(* CODESYS project gprs.lock.20190507.1.project

Project tree, tasks and I/O mapping:
  MIC7001 : Changsha Xiangji-ARM Cortex A9(xilinx zynq7000)-linux, Changsha Xiangji Hiden Technology Co.Ltd, version 3.5.10.40
    application Application
      libraries: Standard, * (System); CAA File, * (CAA Technical Workgroup); CAA Types Extern, * (CAA Technical Workgroup); CAA Callback Extern, * (CAA Technical Workgroup); SysMem, * (System); Util, 3.5.11.0 (System); SysFile, 3.5.9.0 (System); SysTypes Interfaces, * (System); CAN API, 1.0.0.3 (3S - Smart Software Solutions GmbH); AC_DataLog, 3.5.12.0 (3S - Smart Software Solutions GmbH); SysTime, * (System); CAA DTUtil Extern, 3.5.12.0 (CAA Technical Workgroup); CAA SerialCom, 3.5.12.0 (CAA Technical Workgroup); cyber gpio, 3.5.10.40 (cyber)
      task Task_gprs (cyclic, interval 20 ms, priority 10) calls prg_heartbeat
      gprs_lib/
        function block Udp_Config [ST]
        function block reset_gprs [ST]
        function block Udp_Init [ST]
        function block Com_Read [ST]
        function block UDP_Read [ST]
        function block Udp_Write [ST]
      global variables GVL
      GPRS/
        function block fb_get_lac [ST]
        function block fb_get_iccid [ST]
        program prg_heartbeat [ST]
        function block File_Read [ST]
        function block fb_m26 [ST]
        function fn_sn_str_to_byte [ST]
        function Iccid_Get [ST]
        function fn_cyber_layer1 [ST]
        function fn_cyber_userdata200 [ST]
        function fn_cyber_layer2 [ST]
        function fn_cyber_heartBeat [ST]
    SoftMotion General Axis Pool
    IoDrvMIC7001 : IoDrvMIC7001, MyCompany, version 19.1.1
        input  Application.GVL.FR_Protect_DI : BOOL  // Di00-Ai00@C16
        input  Application.GVL.PumpOn_DI : BOOL  // Di01-Ai01@C28
        input  Application.GVL.Remot_Enable_DI : BOOL  // Di02-Ai02@C17
        input  Application.GVL.Rev_PumpOn_DI : BOOL  // Di03-Ai03@C29
        input  Application.GVL.LeftZG_Forward_DI : BOOL  // Di04-Ai04@C30
        input  Application.GVL.Flux_Down_DI : BOOL  // Di05-Ai05@C19
        input  Application.GVL.RightZG_Forward_DI : BOOL  // Di06-Ai06@C31
        input  Application.GVL.ADDOn_DI : BOOL  // Di07-Ai07@C20
        input  Application.GVL.Flux_Up_DI : BOOL  // Di08-Ai08@C18
        input  Application.GVL.Leg_BG_DI : BOOL  // Di09-Ai09@D18
        input  Application.GVL.Limit_Right_DI : BOOL  // Di10-Ai10@D20
        input  Application.GVL.AC_Power_DI : BOOL  // Di11-Ai11@D31
        input  Application.GVL.Limit_Left_DI : BOOL  // Di12-Ai12@D19
        input  Application.GVL.Power_Order_DI : BOOL  // Di14-Ai14@D29
        input  Application.GVL.LeftBG_Forward_DI : BOOL  // Di15-Ai15@D17
        input  Application.GVL.Right_SQ_DI : BOOL  // Di16-Ai16@D28
        input  Application.GVL.RightBG_Forward_DI : BOOL  // Di17-Ai17@D16
        input  Application.GVL.DI_move : BOOL  // Di27-Ai27@C09
        input  Application.GVL.ADDFlux_Down_DI : BOOL  // Di46-Ai46@C22
        input  Application.GVL.ADDFlux_Up_DI : BOOL  // Di47-Ai47@D14
        input  Application.GVL.Motor_Stop_DI : BOOL  // Di48-Pi00@C15
        input  Application.GVL.Motor_Start_DI : BOOL  // Di49-Pi01@C14
        input  Application.GVL.Left_SQ_DI : BOOL  // Di50-Pi02@D22
        input  Application.GVL.Light_Boom_DI : BOOL  // Di51-Pi03@D21
        output Application.GVL.ERR_Power_Order : BOOL  // Do00-Ai18@C25
        output Application.GVL.Remot_Control_DO : BOOL  // Do01-Ai19@C24
        output Application.GVL.Alarm_DO : BOOL  // Do02-Ai20@C13
        output Application.GVL.Light_Boom_DO : BOOL  // Do03-Ai21@C01
        output Application.GVL.DT2_DO : BOOL  // Do04-Ai22@C03
        output Application.GVL.DT3_DO : BOOL  // Do05-Ai23@C04
        output Application.GVL.DT5_DO : BOOL  // Do06-Ai24@C05
        output Application.GVL.DT6_DO : BOOL  // Do07-Ai25@C06
        output Application.GVL.DT4_DO : BOOL  // Do08-Ai26@C08
        output Application.GVL.DT1_DO : BOOL  // Do09-Ai27@C09
        output Application.GVL.Motor_Run_DO : BOOL  // Do10-Ai28@C10
        output Application.GVL.Motor_Start_DO : BOOL  // Do11-Ai29@C11
        output Application.GVL.Horn_Remot_DO : BOOL  // Do24-Ai42@C23
        output Application.GVL.Limit_Left_DO : BOOL  // Do28-Pwmi00@C33
        output Application.GVL.Limit_Right_DO : BOOL  // Do29-Pwmi01@C34
        output Application.GVL.PWM_prop : DWORD  // PWM28-Pwmi00@C33
        output Application.gvl.do_led_run : BOOL  // LED_run
        output Application.gvl.DO_led_err : BOOL  // LED_err
        output Application.gvl.DO_led_usr : BOOL  // LED_usr
        unmapped channels: Ai00@C16, Ai01@C28, Ai02@C17, Ai03@C29, Ai04@C30, Ai05@C19, Ai06@C31, Ai07@C20, Ai08@C18, Ai09@D18, Ai10@D20, Ai11@D31, Ai12@D19, Ai13@D30, Ai14@D29, Ai15@D17, Ai16@D28, Ai17@D16, Ai18-Do00@C25, Ai19-Do01@C24, Ai20-Do02@C13, Ai21-Do03@C01, Ai22-Do04@C03, Ai23-Do05@C04, Ai24-Do06@C05, Ai25-Do07@C06, Ai26-Do08@C08, Ai27-Do09@C09, Ai28-Do10@C10, Ai29-Do11@C11, Ai30-Do12@D34, Ai31-Do13@D35, Ai32-Do14@D23, Ai33-Do15@D12, Ai34-Do16@D10, Ai35-Do17@D09, Ai36-Do18@D08, Ai37-Do19@D07, Ai38-Do20@D05, Ai39-Do21@D04,
          Ai40-Do22@D03, Ai41-Do23@D02, Ai42-Do24@C23, Ai43-Do25@C35, Ai44-Do26@D24, Ai45-Do27@D13, Ai46-Ao00@C22, Ai47-Ao01@D14, Ai48_Pi02, Ai49_Out5V, Ai50_VCC, Ai51_VCC_L, Ai52_VCC_R, Ai53_Pwm-i0, Ai54_Pwm-i1, Ai55_Pwm-i2, Ai56_Pwm-i3, Ai57_CPU-T, Ai58_G-x, Ai59_G-y, Ai60_G-z, Ai61-reserved, Ai62-IO-cntr, Ai63-CDS-cntr, Di13-Ai13@D30, Di18-Ai18@C25, Di19-Ai19@C24, Di20-Ai20@C13, Di21-Ai21@C01, Di22-Ai22@C03, Di23-Ai23@C04, Di24-Ai24@C05, Di25-Ai25@C06, Di26-Ai26@C08, Di28-Ai28@C10, Di29-Ai29@C11, Di30-Ai30@D34, Di31-Ai31@D35, Di32-Ai32@D23, Di33-Ai33@D12,
          Di34-Ai34@D10, Di35-Ai35@D09, Di36-Ai36@D08, Di37-Ai37@D07, Di38-Ai38@D05, Di39-Ai39@D04, Di40-Ai40@D03, Di41-Ai41@D02, Di42-Ai42@C23, Di43-Ai43@C35, Di44-Ai44@D24, Di45-Ai45@D13, Di52-reserved, Di53-reserved, Di54-reserved, Di55-reserved, Di56-reserved, Di57-reserved, Di58-reserved, Di59-reserved, Di60-reserved, Di61-reserved, Di62-reserved, Di63-reserved, Pi00-Di48@C15, Pi01-Di49@C14, Pi02-Di50@D22, Pi03-Di51@D21, Do12-Ai30@D34, Do13-Ai31@D35, Do14-Ai32@D23, Do15-Ai33@D12, Do16-Ai34@D10, Do17-Ai35@D09, Do18-Ai36@D08, Do19-Ai37@D07, Do20-Ai38@D05, Do21-Ai39@D04, Do22-Ai40@D03, Do23-Ai41@D02,
          Do25-Ai43@C35, Do26-Ai44@D24, Do27-Ai45@D13, Do30-Pwmi02@D25, Do31-Pwmi03@D26, PWM00@C25, PWM01@C24, PWM02@C13, PWM03@C01, PWM04@C03, PWM05@C04, PWM06@C05, PWM07@C06, PWM08@C08, PWM09@C09, PWM10@C10, PWM11@C11, PWM12@D34, PWM13@D35, PWM14@D23, PWM15@D12, PWM16@D10, PWM17@D09, PWM18@D08, PWM19@D07, PWM20@D05, PWM21@D04, PWM22@D03, PWM23@D02, PWM24@C23, PWM25@C35, PWM26@D24, PWM27@D13, PWM29-Pwmi01@C34, PWM30-Pwmi02@D25, PWM31-Pwmi03@D26, PWM_I_0@C33, PWM_I_1@C34, PWM_I_2@D25, PWM_I_3@D26,
          Ao00-Ai46@C22, Ao01-Ai47@D14, ctrl_ai_raw, ctrl_adjust, ctrl_adj0, ctrl_adj1, ctrl_adj2, ctrl_adj3, ctrl_adj4
  text list GlobalTextList
*)

// MIC7001/Application/GVL
VAR_GLOBAL
	g_pump_work:BOOL := TRUE;  //液压泵软开关
	g_engine_work:BOOL := TRUE;  //发动机软开关
	
	//小时计相关
	g_running_mins:DINT := 0; //控制器运行的分钟数
	g_machine_start_mins:DINT := 0; //主机出厂时对应的控制器分钟数，需要放在掉电保持的参数区
	g_machine_mins:DINT := 0; //主机运行的分钟数, = g_running_mins - g_machine_start_mins
	g_engine_mins:DINT := 0; //发动机运行的分钟数
	
	g_machine_mins_1_start:DINT := 0; //阶段小时计1开始时间
	g_machine_mins_2_start:DINT := 0; //阶段小时计2开始时间
	
	g_machine_mins_1:DINT := 0;
	g_machine_mins_2:DINT := 0;
	
	// PORT CAN1 GLOBAL HANDLE
	g_hCan1939: CAA.HANDLE ;
	g_hRecv_FEEE: CAA.HANDLE := 0;
	g_hRecv_FEEF: CAA.HANDLE := 0;
	g_hRecv_F003: CAA.HANDLE := 0;
	g_hRecv_F004: CAA.HANDLE := 0;
	g_hRecv_18F: CAA.HANDLE := 0;
	
	//发动机相关实时数据
	g_P_KW_max:DINT := 30;  //当前发动机储备功率
	g_rpm_set: DINT := 1000;  //当前设定转速
	g_rpm_real: DINT := 0; //当前实时转速
	g_fuel_rate_1939:REAL := 0; //从发动机读到的瞬时油耗，单位：ml/s
	g_temp_coolant_1939:REAL := 0; //从发动机读到的水温， 单位：摄氏度
	g_oil_press_1939:REAL := 0; //从发动机读到的机油压力， 单位： kPa
	g_coolant_level_1939:REAL := 0; //从发动机读到的冷却液液位， 单位： 百分比
	g_load_percent_1939:REAL := 0; //从发动机读到的发动机负载率， 单位： 百分比
	g_demand_torque_1939:REAL := 0; //从发动机读到的需求扭矩， 单位： 百分比
	g_real_torque_1939:REAL := 0; //从发动机读到的实际扭矩， 单位：百分比
	
	//统计数据
	g_fuel_depleted: DINT;  //出厂累计油耗，单位：升
	g_fuel_depleted_1: DINT; //阶段一累计油耗，单位：升 
	g_fuel_depleted_2: DINT; //阶段二累计油耗，单位：升
	
	
	g_Eng_Coolaant_Temp:INT;(*spn 110*)
	g_Eng_Fuel_Temp:INT;(*spn 174*)
	g_Eng_Oil_Temp:INT;(*spn 175*)
	g_Turbo_Oil_Temp:INT;(*spn 176*)
	g_Eng_InterCooler_Temp:INT;(*spn 52*)
	g_Eng_InterCooler_Thermostat_Opening:BYTE;(*spn 1134*)
						
	g_res_prop:REAL := 20; //电磁比例阀电阻，动态调整

	//熟数据
	g_ai_press_pump1:REAL;
	g_ai_press_pump1_trace:REAL;
	g_ai_press_pump2:REAL;
	g_ai_press_pump2_trace :REAL;
	g_ai_pilot:REAL;
	g_ai_pilot_trace: REAL;
	g_ai_curr_prop:UINT;
	g_ai_curr_prop_trace:REAL;
	g_ai_oil_water:BOOL;
	g_ai_vcc:DWORD;
	g_ai_fuel_level:REAL;

	g_di_start:BOOL := FALSE; //上电信号
	g_di_move:BOOL := FALSE; //工作装置压力开关
	g_di_work:BOOL := FALSE; //行走压力开关
	g_di_pilot:BOOL := FALSE;  //先导手柄开关输入
	
	g_do_start:BOOL := TRUE;  //启动继电器		
	g_do_ecu:BOOL := TRUE;    //为true为发动机ECU供电
	g_do_pilot:BOOL := FALSE;
	
	g_pwm_prop:DINT := 0; 
	
	g_rpm_trace:REAL := 0;  //示波器变量，转换到0~10之间
	//间接计算数据
	g_psp: REAL := 0;   //电磁比例阀二次压力  MPa
	g_backup_power:REAL := 0;   //发动机储备功率  KW
	g_backup_power_trace:REAL; //示波器变量，转换到0~10之间
	g_duty_power:REAL := 0; //发动机功率利用率
	g_backup_torque:REAL := 0;  //发动机储备扭矩  N*M
	g_backup_torque_trace:REAL;//示波器变量，转换到0~10之间
	g_duty_torque:REAL := 0;  //发动机扭矩利用率
	g_flow1 :REAL := 0;   //前泵流量 L/min
	g_flow1_trace:REAL;//示波器变量，转换到0~10之间
	g_flow2 :REAL := 0;   //后泵流量 L/min
	g_flow2_trace:REAL;//示波器变量，转换到0~10之间
	g_power_pump1 :REAL := 0;   //前泵功率  KW
	g_power_pump1_trace:REAL;//示波器变量，转换到0~10之间
	g_power_pump2 :REAL := 0;   //后泵功率  KW
	g_power_pump2_trace:REAL;//示波器变量，转换到0~10之间
	g_torque_pump1 :REAL := 0;  //前泵输出扭矩  N*M
	g_torque_pump2 :REAL := 0;  //后泵输出扭矩  N*M
	
// I/O port mapping var
	AI_pump1:DWORD; //前泵压力
	AI_pump2:DWORD; //后泵压力
	AI_pilot:DWORD; //先导压力
	AI_curr_prop:DWORD; //电磁比例阀电流
	AI_oil_water:DWORD; //油水分离器
	AI_vcc:DWORD; //电源电压 mV
	AI_grade:DWORD; //油门旋钮
	AI_temp_oil:DWORD; //液压油温
	AI_fuel_level:DWORD; //液位传感器
		
	
	DI_start: BOOL; //启动信号
	DI_pilot:BOOL; //先导手柄闭合
	DI_move:BOOL; //行走压力开关
	DI_work:BOOL; //作业压力开关
	DI_air_filter:BOOL;  //空滤堵塞
	DI_idle_button:BOOL;  //机械怠速按钮
	DI_high_power:BOOL; //增力信号输入
	
	
	DO_start: BOOL := FALSE; //驱动启动电机
	DO_stop: BOOL := TRUE;  //驱动熄火继电器
	DO_pilot :BOOL := TRUE;  //驱动先导阀
	DO_high_power:BOOL := FALSE; //增力输出
	DO_high_speed:BOOL := FALSE; //高速输出
	DO_dump_load:BOOL := FALSE; //卸载输出
	
					
	PWM_prop:DWORD; //油泵电磁比例阀	
	
	RPM_engine:UINT; //柴油机转速  J1939

	DO_led_run:BOOL;
	DO_led_err:BOOL;
	DO_led_usr:BOOL;
	
// 档位校准	
	adj_gear: BOOL := FALSE;  //校准档位旋钮
	gear_grade: UINT := 1;   //档位旋钮对应的档位
	running_grade:UINT := 1;  //当前实际运行的档位
	
	g_grade: DINT;	  //发动机档位
	//各档位对应的转速
	grade_rpm : ARRAY [1..10] OF DINT := [1200, 1350, 1450, 1550, 1650, 1750, 1850, 1950, 2050, 2200];
	
	//各档位对应的旋钮采样值（mV）
	grade_mv: ARRAY[1..10] OF DINT := [1534, 1705, 1876, 2056, 2242, 2439, 2625, 2810, 2988, 3168];

//显示屏发送来的命令
	cmd_auto_idle : BOOL := FALSE;
	cmd_high_speed: BOOL := FALSE;	
	cmd_more_power: BOOL := FALSE;
	cmd_clear_hours : BOOL := FALSE;
	cmd_clear_hours_1 :BOOL := FALSE;
	cmd_clear_hours_2 :BOOL := FALSE;
	
	//各模式的比例阀电流值
	pwm_of_mode_h : DINT := 580;  //H模式
	pwm_of_mode_s : DINT := 520;  //S模式
	pwm_of_mode_l : DINT := 490;  //L模式
	
	C_RPM_MIN: DINT := 800;
	C_RPM_IDLE: DINT := 1450;
	C_RPM_MAX : DINT := 2300;
	
	C_H_MAX_RPM: DINT := 2200;
	C_S_MAX_RPM: DINT := 2050;
	C_L_MAX_RPM: DINT := 1900;
	
	g_time_good: BOOL := FALSE;  //控制器本地时钟校准完成
	
	remote_data00:BYTE;
	remote_data01:BYTE;
	remote_data02:BYTE;
	remote_data03:BYTE;
	remote_data04:BYTE;
	remote_data05:BYTE;
	remote_data06:BYTE;
	remote_data07:BYTE;
	remote_data08:BYTE;
	remote_data09:BYTE;
	remote_data010:BYTE;
	remote_data011:BYTE;
	remote_data012:BYTE;
	
	Parameter_Page_default:BOOL;
	Flux_Init:BOOL;
	INIT_SUCC:BOOL;     //常闭
	Work_Time_S:DINT;
	Work_Time_M:DINT;
	Work_Time_H:DINT;
	TON_Work_Time:ton;
	Work_Time_Old:DINT;
	Work_Time_All:DINT;
	TON_Work_Store:ton;
	Work_Store:BOOL;
	F_Trig_Pump_Start:f_trig;
	R_Trig_SQ:r_trig;
	bR_Direction_exchange:BOOL;
	sR_Direction_exchange_Count:DINT;
	Timer_Pump_1Counter:DINT;
	TON_Direction_exchange:ton;
	Timer_Pump_11Counter:REAL;
	Pump_Counter:REAL;
	Diameter:REAL;          //混凝土缸直径*)
	Length:REAL;           //主缸行程
	Cube_Meter_Pump:REAL;  //泵送实时排量
	ADD_Setting_Temp:DINT;
	ADD_Setting:DINT;
	ADD_TEMPA:REAL;
	ADD_TEMPK:REAL;
	ADDFlux_Up_DI:BOOL;        //本地速凝剂+
	ADDFlux_Up_Remot_DI:BOOL;  //远程速凝剂+
	ADDFlux_Down_DI:BOOL;      //本地速凝剂-
	ADDFlux_Down_Remot_DI:BOOL;//远程速凝剂-
	ADD_Setting_Adjust:DINT;
	ADD_in_Coment_All:REAL;
	DT9_PWM:DINT;
	PUMP_Current_OUT:DINT;         //泵送电流输出值
	Power_Order_DI:BOOL;           //相序错误输入
	ERR_Power_Order:BOOL;          //相序错误指示灯
	RS_Motor_Start:RS;
	TON_Motor_Start:ton;
	TOF_Motor_Start:tof;
	Motor_Start_DI:BOOL;          //电机启动信号
	Motor_Stop_DI:BOOL;           //电机停止信号
	Estop_Remot_DI:BOOL;          //遥控急停开关
	Estop_Manul_DI:BOOL;          //料斗急停开关
	Motor_Start_DO:BOOL;          //电机星型运转
	Motor_Run_DO:BOOL;            //电机三角形运转
	Light_Boom_DI:BOOL;             //臂架照明开关
	Light_Boom_remote_DI:BOOL;             //臂架照明开关
	Light_Boom_DO:BOOL;             //臂架照明继电器
	Remot_Enable_DI:BOOL;          //遥控-就地切换开关
	Remot_Control_DO:BOOL;         //遥控-就地指示灯
	


	Boom_Enable_DI:BOOL;        //臂架动作使能信号
	Limit_Left_DI:BOOL;        //臂架左限位
	Limit_Right_DI:BOOL;       //臂架右限位
	Limit_Left_DO:BOOL;        //臂架左限位输出
	Limit_Right_DO:BOOL;       //臂架右限位输出
	ADDOn_Remot_DI:BOOL;       //速凝剂远程启动输入
	ADD_DO:BOOL;               //速凝剂启动输出
	ADDOn_DI:BOOL;             //速凝剂本地启动输入
	Leg_Move_DI:BOOL;
	Leg_BG_DI:BOOL;           //臂架-支腿切换输入
	
	Horn_Remot_DI:BOOL;
	Horn_Remot_DO:BOOL;	
	
	Flux_Up_DI:BOOL;         //本地泵送排量+
	Flux_Up_Remot_DI:BOOL;   //远程泵送排量+
	Flux_Down_DI:BOOL;       //本地泵送排量-
	Flux_Down_Remot_DI:BOOL; //远程泵送排量-
	Flux_Setting:DINT;       //泵送排量调节中间变量
	Pump_On:BOOL;          //正泵输出信号
	Rev_Pump_On:BOOL;      //反泵输出信号
	PumpOn_DI:BOOL;        //本地正泵输入
	PumpOn_Remot_DI:BOOL; //远程正泵输入
	Rev_PumpOn_DI:BOOL;   //本地反泵信号
	Rev_PumpOn_Remot_DI:BOOL;  //远程反泵
	Pump_Start:BOOL;          //泵送启动
	R_Pump:R_TRIG;
	Pump_Init:BOOL;
	Pump_ADD_V:REAL;      //泵送累计方量
	Pump_ADD_once:REAL:=0;   //当次泵送方量
	SQ1:BOOL;             //左限位
	SQ2:BOOL;             //右限位
	R_Pump_c:R_TRIG;
	
	Right_Forward:BOOL;
	Left_Forward:BOOL;
	Delay_Time:TIME;
	TON_T_Exchange:ton;
	TON_SQ1:ton;
	TON_SQ2:ton;
	Permit_Exchange:BOOL;
	
	T_Exchange:BOOL;
	     
	
	LeftZG_Forward_DI:BOOL;  //主缸左输入
	RightZG_Forward_DI:BOOL; //主缸右输入
	LeftBG_Forward_DI:BOOL;  //摆缸左输入
	RightBG_Forward_DI:BOOL; //摆缸右输入

    Left_SQ_DI:BOOL;       //左限位开关
	Right_SQ_DI:BOOL;      //右限位开关	
	
	DT1_DO:BOOL;               //臂架减压阀
	DT2_DO:BOOL;      //主缸左
	DT3_DO:BOOL;      //主缸右
	DT4_DO:BOOL;      //支腿-摆缸建压
	DT5_DO:BOOL;       //摆缸左
	DT6_DO:BOOL;      //摆缸右
	
	
	
	AI_dbzz:BYTE;
	AI_dbfz:BYTE;
	AI_dbf:BYTE;
	AI_dby:BYTE;

	AI_xbf:BYTE;
	AI_xby:BYTE;
	AI_xbsc:BYTE;
	AI_xbsh:BYTE;

    AI_pzzz:BYTE;
	AI_pzfz:BYTE;
	AI_pzf:BYTE;
	AI_pzy:BYTE;

	AI_sd:BYTE;
	
	remote_DI_1:BYTE;
	remote_DI_2:BYTE;
	
	
    BOOM_pwm_dbzz:DWORD;          //大臂正转
	BOOM_pwm_dbfz:DWORD;          //大臂反转
	BOOM_pwm_dbf:DWORD;           //大臂俯
	BOOM_pwm_dby:DWORD;           //大臂仰
	
	BOOM_pwm_xbf:DWORD;           //小臂俯
	BOOM_pwm_xby:DWORD;           //小臂仰
	BOOM_pwm_xbsc:DWORD;          //小臂伸
	BOOM_pwm_xbsh:DWORD;          //小臂缩
	
	BOOM_pwm_pzzz:DWORD;          //喷嘴正转
	BOOM_pwm_pzfz:DWORD;          //喷嘴反转
	BOOM_pwm_pzf:DWORD;           //喷嘴俯
	BOOM_pwm_pzy:DWORD;           //喷嘴仰
		
	BOOM_pwm_sd:DWORD;          //刷动

	snj_pwm:DWORD;               //速凝剂排量调节
	DT8_PWM:DINT;              //泵送排量调节
	
	Current_Max_dbzz:INT;       //大臂正转最大电流
	Current_Min_dbzz:INT;       //大臂正转最小电流
	Current_Max_dbfz:INT;       //大臂反转最大电流
	Current_Min_dbfz:INT;       //大臂反转最小电流
	Current_Max_dbf:INT;       //大臂俯最大电流
	Current_Min_dbf:INT;       //大臂俯最小电流
	Current_Max_dby:INT;       //大臂仰最大电流
	Current_Min_dby:INT;       //大臂仰最小电流
	
	Current_Max_xbf:INT;       //小臂俯最大电流
	Current_Min_xbf:INT;       //小臂俯最小电流
	Current_Max_xby:INT;       //大臂仰最大电流
	Current_Min_xby:INT;       //大臂仰最小电流
	Current_Max_xbsc:INT;       //小臂伸出最大电流
	Current_Min_xbsc:INT;       //小臂伸出最小电流
	Current_Max_xbsh:INT;       //小臂缩回最大电流
	Current_Min_xbsh:INT;       //小臂缩回最小电流
	
	Current_Max_pzzz:INT;       //喷嘴正转最大电流
	Current_Min_pzzz:INT;       //喷嘴正转最小电流
	Current_Max_pzfz:INT;       //喷嘴反转最大电流
	Current_Min_pzfz:INT;       //喷嘴反转最小电流
	Current_Max_pzf:INT;       //喷嘴俯最大电流
	Current_Min_pzf:INT;       //喷嘴俯最小电流
	Current_Max_pzy:INT;       //喷嘴仰个最大电流
	Current_Min_pzy:INT;       //喷嘴仰最小电流
	
	Current_Max_sd:INT;       //刷动最大电流
	Current_Min_sd:INT;       //刷动最小电流
	
	
	

	Parameter_interRatain: ARRAY [0..25] OF DINT;
	Parameter_Page_Change :BOOL;
	SYMC_Version_Main:SINT;
	SYMC_Version_Sub:SINT;
	PUMP_Current_Min:DINT;         //泵送最小电流
	PUMP_Current_Max:DINT;        //泵送最大电流
	PUMP_Current_Init:DINT;       //泵送初始电流
	Rate_pump:REAL;                       //泵送吸料率
	interRetain_DINT:DINT;
	PUMP_Current_Min_default:DINT;     //泵送最小排量
	PUMP_Current_Max_default:DINT;     //泵送最大排量
	Density_of_ADD_default:REAL;      //速凝剂比重
	Coment_Per_M3_default:DINT;      //混凝土水泥含量
	Rate_pump_default:REAL;          //泵送吸料率
	Phase_Protect_default:BOOL;
	
	ADD_Adjust:REAL;
	ADD_Adjust_default:REAL;
	
	PUMP_Current_Init_default:DINT;
	ADD_in_Coment_Min:REAL;
	ADD_in_Coment_Max:REAL;
	ADD_Min_out:BYTE;     //速凝剂最小档位
	ADD_Max_out:BYTE;     //速凝剂最大档位
	ADD_in_Coment_default:BYTE;     //速凝剂初始比
	ADD_OUT:BYTE;        //速凝剂输出档位
	ADD_rate:BYTE;       //速凝剂系数
	
	
	TON_Work_Time1:ton;

//面板通讯//



	

Change_Save_DINT:DINT;
Cylinder_Diameter:REAL;        //液压缸内径*)
Cylinder_Piston_Diameter:REAL; //活塞杆直径*)
Speed_Motor:REAL;             //电机转速
Q_Oil_Pump:REAL;              //实际流量*)
Capacity_Oil_Pump:REAL;      //实际排量输出，130为满排量
Counter_Pump:REAL;      //换向次数
Cube_Onetime:REAL;      //单词泵送方量
R_Flux_Up:r_trig;
R_Flux_Down:r_trig;
ADD_PWM_Adjust:DINT;
R_ADDFlux_Up:r_trig;
R_ADDFlux_Down:r_trig;

ERR_SQ1:BOOL;
ERR_SQ2:BOOL;
Send_Buff2:ARRAY[0..7] OF BYTE;
RC_Recive_SINT5:SINT;
RC_Recive_SINT4:SINT;
Alarm_DO:BOOL;               //故障报警
TON_SQ1_ERR1:ton;
TON_SQ1_ERR2:ton;
TON_SQ2_ERR1:ton;
TON_SQ2_ERR2:ton;
ceshi1:SINT;
ceshi2:SINT;
ceshi4:SINT;
ceshi5:SINT;
ceshi3:DINT;
send_test:DINT;
TON_Save_Recive:ton;
Can_Recive_P1:DINT;
CAN_Recive_Buff:ARRAY[0..23] OF BYTE;
CAN_Recive:DINT;
Rate_pump_TEST:REAL;
PUMP_Current_Min_TEST:DINT;
PUMP_Current_Max_TEST:DINT;
PUMP_Current_Init_TEST:DINT;
Density_of_ADD_TEST:REAL;
Coment_Per_M3_TEST:DINT;
ADD_in_Coment_TEST:REAL;
ADD_in_Coment_Min_TEST:REAL;
ADD_in_Coment_Max_TEST:REAL;
ADD_Adjust_TEST:REAL;
Can_Send_P2:DINT;
CHANGE1:DINT;
CHANGE2:DINT;
CHANGE3:DINT;
CHANGE4:DINT;
Parameter_Page_default_TEST:BOOL;
can_test1:BOOL;
can_test2:BOOL;
can_test3:BOOL;
can_test4:BOOL;
can_test5:BOOL;
can_test6:BOOL;

F_TRIG_Stop:f_trig;
PUMP_Current_OUT_TEMP:DINT;
R_TRIG_ADDON:r_trig;
TOF_R_ADDON:tof;
F_Trig_MotorRun_DO:f_trig;

Motor_Time_S:DINT;
Motor_Time_M:DINT;
Motor_Time_H:DINT;
Motor_Time_All:DINT;
Motor_Time_Old:DINT;
Work_Store1:BOOL;
Lost_Time:DINT;
Lock_ID_300:SINT;
Password:DINT;
Display_Lock_300H:BOOL;
Display_ID:DINT;
Display_Lock_500H:BOOL;
Enable_NOLock_Machine:BOOL;
Ton_Password_Move:ton;
Ton_Password_Move11:ton;
OK_Open_Lock:BOOL;
Recive_Buff2:ARRAY[0..7] OF BYTE;
Recive_Buff3:ARRAY[0..7] OF BYTE;
TOF_R_NOLock_Machine:tof;
TON_Delay_Left:ton;
TON_Delay_Right:ton;
OK_Open_Lock_test:BOOL;
Lost_time_send:DINT;
Enable_Lock_Machine_test:SINT;
Enable_NOLock_Machine_test:BOOL;
R_Enable_Lock:r_trig;
AC_Power_DI:BOOL;                   //交流电源输入
TEST_LOCK:BOOL;
DINT_TEST_LOCK1:DINT;
DINT_TEST_LOCK2:DINT;
DINT_TEST_LOCK3:DINT;
DINT_TEST_LOCK4:DINT;
R_Lock_Machine:r_trig;
Password_NOlock_Machine:BOOL;
Display_Lock_10M:BOOL;
Display_Lock_100H:BOOL;
Lock10M_Machine:BOOL;
Lock_time_add1:DINT;
Password_10:DINT;
Password_100:DINT;
Lock_time_add:DINT;
Lock100H_Machine:BOOL;
Password_300:DINT;
Lock300H_Machine:BOOL;
Lock500H_Machine:BOOL;
Password_500:DINT;
Password_NOlock:DINT;
Display_Lock_Move:BOOL;
Lost_Time1:DINT;
R_Open_Machine:r_trig;
OK_Open_Machine:BOOL;
Enable_N0Lock_Machine:BOOL;
LOCK_Store:BOOL;
test_1116:BOOL;
DINT_TEST_LOCK5:DINT;
DINT_TEST_LOCK6:DINT;
TEST_11116:BOOL;
TEST_11117:BOOL;
TEST_11118:BOOL;
TEST_11119:BOOL;
TEST_11120:BOOL;
TEST_11121:BOOL;
TEST_11122:BOOL;
TEST_11123:BOOL;
LOCK_Store1:BOOL;
LOCK_Store2:BOOL;
LOCK_Store3:BOOL;
LOCK_Store4:BOOL;
LOCK_Store5:BOOL;
LOCK_Store6:BOOL;
TEST_1111111117:BOOL;
Lock10M_TEST:BOOL;
Lock100H_TEST:BOOL;
Lock300H_TEST:BOOL;
Lock500H_TEST:BOOL;
Password_NOlock_TEST:BOOL;
FR_Protect_DI:BOOL;

	
	
END_VAR

VAR_GLOBAL CONSTANT
	inmode_file:STRING:='in_mode.txt';
	mins_file :STRING := '/userapp/r_mins.txt';
END_VAR

// MIC7001/Application/GPRS/prg_heartbeat
PROGRAM prg_heartbeat
VAR_OUTPUT
	lock_state :INT := 0;
	unlock_state :INT := 0;
	lock_unlock_level :INT := 0;
	delay_time :INT := 0;
END_VAR

VAR
	is_inited :BOOL := FALSE;
	g_m26:fb_m26;
	udp_handle :CAA.HANDLE; 
	udp_write_fb:Udp_Write;
	udp_read_fb:Udp_Read;
	file_read_fb:File_Read;
	com_read_fb :Com_Read;


	size :CAA.SIZE;	
	Writebuffer: 			ARRAY[1..200] OF BYTE;
	Readbuffer: 			ARRAY[0..1499] OF BYTE;
	ReadbufferStr: STRING;
	atcState :INT := 0;
	
	writeUdpState :INT := 0;
	readUdpState :INT := 0;
	
	i :INT;
	count :INT := 0;
	
	rtc_fb: RTC;
	dtu_set_dt_fb: dtu.SetDateAndTime;
	
	sn_file_name :STRING := '/userapp/sn.txt';
	time_file_name :STRING := '/userapp/r_mins.txt';
	is_read :BOOL := FALSE;
	read_count :INT := 0;
	readFileState :INT := 0;
	ton_fb :TON;
	iccid_read_buffer :STRING;
	position :INT := -1;
	new_date:DT;
	get_iccid:fb_get_iccid;
	get_lac:fb_get_lac;
	iStat :UINT := 0;
	lac : STRING(4) := '0000';
	ci : STRING(4) := '0000';
	lenHearBeat:UINT;
	dataHearBeat:ARRAY[0..255] OF BYTE;
	ton_hb:ton; //heartbeat timer 
	bReturn:BOOL;
	lenLayer2:UINT;
	dataLayer2:ARRAY[0..255] OF BYTE;
	lenLayer1:UINT;
	lenRecvLayer1:UINT := 1500;
	dataLayer1:ARRAY[0..255] OF BYTE;
	bSN :ARRAY[0..6] OF BYTE;
	sub_str:STRING(8);
	num :UINT;
	lenHeartBeat: UINT;
	sn: STRING;
	work_time: UDINT;
	dataIndex :UINT := 0;
	cntr_lac:UINT := 0;
	cntr_iccid:UINT := 0;
	
	recv_size :CAA.SIZE;
	
	cntr_user_data:UINT := 0;
	lenUserData:UINT;
	dataUserData:ARRAY[0..255] OF BYTE;
END_VAR

CASE iStat OF
0:
	g_m26(enable := TRUE, ipaddr := '47.107.240.29', port := 34567);  //共用的基础模块，只要有一个地方调用即可	
	IF g_m26.xDone THEN
		iStat := 1;
	END_IF


1:  // read iccid
	get_iccid(xExecute := FALSE);
	iStat := 2;
	cntr_iccid := 0;
	
2:
	get_iccid(xExecute := TRUE, m26_handle := g_m26.handle_m26);
	IF get_iccid.xDone THEN
		iccid_read_buffer := get_iccid.iccid;
		iStat := 10;
	END_IF
	cntr_iccid := cntr_iccid + 1;
	IF cntr_iccid > 600 THEN   // 1 min
		iStat := 1;
	END_IF
	
10: //read sn
	file_read_fb(file_name := sn_file_name);
	IF file_read_fb.isRead THEN
		sn := file_read_fb.sReadLine;
		iStat := 15;
	END_IF
	
15:
	get_lac(xExecute := FALSE);	
	iStat := 20;
	cntr_lac := 0;
	
20:
	get_lac(xExecute := TRUE, m26_handle := g_m26.handle_m26);
	IF get_lac.xDone THEN
		lac := get_lac.lac;
		ci := get_lac.ci;
		iStat := 30;
	END_IF
	cntr_lac := cntr_lac + 1;
	IF cntr_lac > 200 THEN
		iStat := 0;
	END_IF
	
30:
	file_read_fb(file_name := time_file_name);
	IF file_read_fb.isRead THEN
		work_time := STRING_TO_UDINT(file_read_fb.sReadLine);
		iStat := 100;
	END_IF
	
100:
	ton_fb(IN := TRUE, PT := T#10S);
	IF (ton_fb.Q) THEN
		ton_fb(IN := FALSE, PT := T#10S);
		iStat := 200;
	END_IF
	
200:
	bReturn := fn_cyber_heartBeat(	  //填充第三层：心跳帧
						lac_str := lac, 
						cid_str := ci, 
						ccid_str := iccid_read_buffer, 
						mins := work_time, 
						clientCode := 8, 
						machineCode := 9, 
						pLenOut := ADR(lenHearBeat), 
						pDataOut := ADR(dataHearBeat));
	IF NOT bReturn THEN
		RETURN;
	ELSE
		iStat := 300;
	END_IF;

300:
	dataIndex := dataIndex + 1;
	bReturn := fn_cyber_layer2( //填充第二层，数据层
						dataType := 1,
						paraId := 0,
						dataIndex := dataIndex,
						ver := 1,
						res1 := 0,
						LenIn := lenHearBeat,
						pDataIn := ADR(dataHearBeat),
						pLenOut := ADR(lenLayer2),
						pDataOut := ADR(dataLayer2));
						
	IF NOT bReturn THEN
		RETURN;
	ELSE
		iStat := 400;
	END_IF;
	
400:
	bSN := fn_sn_str_to_byte(sn);
	bReturn := fn_cyber_layer1(    //填充第一层，设备层
						sn := ADR(bSN),
						ver := 1,
						lenIn := lenLayer2,
						pDataIn := ADR(dataLayer2),
						pLenOut := ADR(lenLayer1),
						pDataOut := ADR(dataLayer1));
	IF NOT bReturn THEN
		RETURN;
	ELSE
		udp_write_fb(xExecute := FALSE);
		iStat := 500;
	END_IF;
		
	
500:
	udp_write_fb(xExecute := TRUE, com := g_m26.handle_m26, buffer := ADR(dataLayer1), size := lenLayer1);
	IF udp_write_fb.xDone THEN
		udp_write_fb(xExecute := FALSE);
		udp_read_fb(xExecute := FALSE);
		cntr_user_data := cntr_user_data + 1;
		IF cntr_user_data > 10 THEN
			cntr_user_data := 0;
			iStat := 550;  // 每发10次心跳，发送一次自定义数据,可自行定义
		ELSE
			iStat := 600; 
		END_IF
	END_IF
	
	IF udp_write_fb.xError THEN  
		udp_write_fb(xExecute := FALSE);
		iStat := 15; 
	END_IF

550:  //发送用户自定义数据
	fn_cyber_userdata200(  //填充第三层，用户数据
		data0 := 16#01020304,     //主机工作时间（分钟数）,请用实际变量代替
		data1 := 16#05060708,     //工作方量（方）,请用实际变量代替
		data2 := 0,     //预留作以后添加
		data3 := 0,  			
		data4 := 0,
		data5 := 0,
		data6 := 0,
		data7 := 0,
		
		pLenOut := ADR(lenUserData),
		pDataOut := ADR(dataUserData));
		
		dataIndex := dataIndex + 1;
		fn_cyber_layer2( //填充第二层，数据层
						dataType := 1,   //1： 重复发送，无需应答的过程数据
						paraId := 200,  //200:用户自定义数据
						dataIndex := dataIndex,
						ver := 1,
						res1 := 0,
						LenIn := lenUserData,
						pDataIn := ADR(dataUserData),
						pLenOut := ADR(lenLayer2),
						pDataOut := ADR(dataLayer2));
						
		fn_cyber_layer1(    //填充第一层，设备层
						sn := ADR(bSN),
						ver := 1,
						lenIn := lenLayer2,
						pDataIn := ADR(dataLayer2),
						pLenOut := ADR(lenLayer1),
						pDataOut := ADR(dataLayer1));			
		iStat := 560;
560:
	udp_write_fb(xExecute := TRUE, com := g_m26.handle_m26, buffer := ADR(dataLayer1), size := lenLayer1);
	IF udp_write_fb.xDone THEN
		udp_write_fb(xExecute := FALSE);
		iStat := 600;
	END_IF
	
	IF udp_write_fb.xError THEN  
		udp_write_fb(xExecute := FALSE);
		iStat := 15; 
	END_IF
600:
	udp_read_fb(xExecute := TRUE, com := g_m26.handle_m26, buffer := ADR(Readbuffer), rsize := SIZEOF(Readbuffer));
	IF udp_read_fb.xDone THEN  //接收到数据
	 	recv_size := udp_read_fb.size;
		udp_read_fb(xExecute := FALSE);
		iStat := 15; //read mins and lca again
		IF recv_size = 26 THEN
			lock_state := BYTE_TO_INT(Readbuffer[20]);
			unlock_state := BYTE_TO_INT(Readbuffer[21]);
			lock_unlock_level := BYTE_TO_INT(Readbuffer[22]);
			delay_time := BYTE_TO_INT(Readbuffer[23]);
		END_IF
	END_IF
	
	IF udp_read_fb.xError THEN  //接收到数据
		udp_read_fb(xExecute := FALSE);
		recv_size := 0;
		iStat := 15; //read mins and lca again
	END_IF

END_CASE

RETURN;

END_PROGRAM

// MIC7001/Application/GPRS/fn_cyber_heartBeat
FUNCTION fn_cyber_heartBeat : bool
VAR_INPUT
	lac_str:STRING(4);
	cid_str:STRING(4);
	ccid_str:STRING(21);
	mins:UDINT;
	clientCode:UINT;
	machineCode:UINT;
	pLenOut:POINTER TO UINT;
	pDataOut:POINTER TO BYTE;
END_VAR
VAR
	index: UINT;
	data_uint: UINT;
	data_byte_array:ARRAY[0..9] OF BYTE;
	i: INT;
END_VAR

fn_cyber_heartBeat := FALSE;

index := 0;
data_uint := STRING_TO_UINT(concat('16#',lac_str));
pDataOut[index] := ANY_TO_BYTE(data_uint/256);
index := index + 1;

pDataOut[index] := ANY_TO_BYTE(data_uint MOD 256);
index := index + 1;

data_uint := STRING_TO_UINT(concat('16#',cid_str));
pDataOut[index] := ANY_TO_BYTE(data_uint/256);
index := index + 1;

pDataOut[index] := ANY_TO_BYTE(data_uint MOD 256);
index := index + 1;

data_byte_array := Iccid_Get(ccid_str);
FOR i := 0 TO 9 DO
	pDataOut[index] := data_byte_array[i];
	index := index + 1;
END_FOR

pDataOut[index] := ANY_TO_BYTE(mins/256/256/256);
index := index + 1;

pDataOut[index] := ANY_TO_BYTE(mins/256/256);
index := index + 1;

pDataOut[index] := ANY_TO_BYTE(mins/256);
index := index + 1;

pDataOut[index] := ANY_TO_BYTE(mins);
index := index + 1;

pDataOut[index] := ANY_TO_BYTE(clientCode/256);
index := index + 1;

pDataOut[index] := ANY_TO_BYTE(clientCode);
index := index + 1;

pDataOut[index] := ANY_TO_BYTE(machineCode/256);
index := index + 1;

pDataOut[index] := ANY_TO_BYTE(machineCode);
index := index + 1;

pLenOut^ := index;

fn_cyber_heartBeat := TRUE;

END_FUNCTION

// MIC7001/Application/GPRS/Iccid_Get
FUNCTION Iccid_Get : ARRAY[0..9] OF BYTE
VAR_INPUT
	iccd :STRING;
END_VAR
VAR
	iccid_code :ARRAY[0..9] OF BYTE;
	
	byteHigh :BYTE := 0;
	byteLow :BYTE := 0;
	dstLen :INT := 0;
	
	srcIndex :INT := 0;
	bytesIndex :INT := 0;
	sub_str:STRING(32);
END_VAR

dstLen := len(iccd) / 2;

sub_str := iccd;
FOR bytesIndex := 0 TO dstLen - 1 DO
	iccid_code[bytesIndex] := BYTE_TO_BCD(STRING_TO_BYTE(left(sub_str,2)));	
	sub_str := delete(sub_str,2,1);
END_FOR

Iccid_Get := iccid_code;

END_FUNCTION

// MIC7001/Application/GPRS/fn_cyber_layer2
FUNCTION fn_cyber_layer2 : bool
VAR_INPUT
	dataType : BYTE := 0;
	paraId :BYTE := 0;
	dataIndex : UINT := 0;
	ver :BYTE := 1;
	res1 :BYTE := 0;
	LenIn :UINT := 0;
	pDataIn :POINTER TO BYTE;
	pLenOut :POINTER TO UINT;
	pDataOut :POINTER TO BYTE;
END_VAR
VAR
	i:UINT:= 0;
	index:UINT := 0;
END_VAR

fn_cyber_layer2 := FALSE;

index := 0;
pDataOut[index] := dataType;
index := index + 1;

pDataOut[index] := paraId;
index := index + 1;

pDataOut[index] := ANY_TO_BYTE(dataIndex/256);
index := index + 1;

pDataOut[index] := ANY_TO_BYTE(dataIndex MOD 256);
index := index + 1;

pDataOut[index] := ver;
index := index + 1;

pDataOut[index] := res1;
index := index + 1;

pDataOut[index] := ANY_TO_BYTE(LenIn/256);
index := index + 1;

pDataOut[index] := ANY_TO_BYTE(LenIn MOD 256);
index := index + 1;

FOR i := 0 TO LenIn-1 DO
	pDataOut[index] := pDataIn[i];
	index := index + 1;
END_FOR

pLenOut^ := index;

fn_cyber_layer2 := TRUE;
RETURN;

END_FUNCTION

// MIC7001/Application/GPRS/fn_sn_str_to_byte
FUNCTION fn_sn_str_to_byte : ARRAY[0..6] OF BYTE
VAR_INPUT
	sn:STRING(16);
END_VAR
VAR
	i: INT;
	bSN: ARRAY[0..6] OF BYTE;
	sub_str: STRING(255);
	num: UINT;
	bcd: UINT;
END_VAR

// 1.2 12
sub_str := mid(sn, 2, 4);
bcd := STRING_TO_UINT(sub_str);
bcd := (bcd / 10) *16 + (bcd MOD 10);
bSN[0] := UINT_TO_BYTE(bcd);

// 1.3 34
sub_str := mid(sn, 2, 6);
bcd := STRING_TO_UINT(sub_str);
bcd := (bcd / 10) *16 + (bcd MOD 10);
bSN[1] := UINT_TO_BYTE(bcd);

// 1.4 56
sub_str := mid(sn, 2, 8);
bcd := STRING_TO_UINT(sub_str);
bcd := (bcd / 10) *16 + (bcd MOD 10);
bSN[2] := UINT_TO_BYTE(bcd);

// 1.5 78
sub_str := mid(sn, 2, 10);
bcd := STRING_TO_UINT(sub_str);
bcd := (bcd / 10) *16 + (bcd MOD 10);
bSN[3] := UINT_TO_BYTE(bcd);

// 1.6 1234
sub_str := mid(sn, 2, 12);
bcd := STRING_TO_UINT(sub_str);
bcd := (bcd / 10) *16 + (bcd MOD 10);
bSN[4] := UINT_TO_BYTE(bcd);

sub_str := mid(sn, 2, 14);
bcd := STRING_TO_UINT(sub_str);
bcd := (bcd / 10) *16 + (bcd MOD 10);
bSN[5] := UINT_TO_BYTE(bcd);

fn_sn_str_to_byte := bSN;

END_FUNCTION

// MIC7001/Application/GPRS/fn_cyber_layer1
FUNCTION fn_cyber_layer1 : bool
VAR_INPUT
	sn:POINTER TO BYTE;
	ver:BYTE := 0;
	lenIn:UINT := 0;
	pDataIn:POINTER TO BYTE;
	pLenOut:POINTER TO UINT ;
	pDataOut: POINTER TO BYTE;
END_VAR
VAR
	i:UINT;
	index:UINT;
	checksum:UINT;
	res1 :BYTE := 0;
END_VAR

fn_cyber_layer1 := FALSE;

index := 0;
checksum := 0;
FOR i := 0 TO 5 DO
	pDataOut[index] := sn[i];
	index := index+1;
	checksum := checksum + sn[i];
END_FOR

pDataOut[index] := ver;
index := index+1;
checksum := checksum + ver;

pDataOut[index] := res1;
index := index+1;
checksum := checksum + res1;

pDataOut[index] := res1;
index := index+1;
checksum := checksum + res1;

pDataOut[index] := res1;
index := index+1;
checksum := checksum + res1;

pDataOut[index] := ANY_TO_BYTE(lenIn/256);
index := index+1;
checksum := checksum + ANY_TO_BYTE(lenIn/256);

pDataOut[index] := ANY_TO_BYTE(lenIn MOD 256);
index := index+1;
checksum := checksum + ANY_TO_BYTE(lenIn MOD 256);

FOR i := 0 TO lenIn-1 DO
	pDataOut[index] := pDataIn[i];
	index := index+1;	
	checksum := checksum + pDataIn[i];
END_FOR

pDataOut[index] := ANY_TO_BYTE(checksum/256);
index := index+1;

pDataOut[index] := ANY_TO_BYTE(checksum MOD 256);
index := index+1;

pLenOut^ := index;

fn_cyber_layer1 := TRUE;

END_FUNCTION

// MIC7001/Application/GPRS/fn_cyber_userdata200
FUNCTION fn_cyber_userdata200 : BOOL  //发送8个4字节的用户自定义数据到云端
VAR_INPUT
	data0:UDINT;
	data1:UDINT;
	data2:UDINT;
	data3:UDINT;
	data4:UDINT;
	data5:UDINT;
	data6:UDINT;
	data7:UDINT;
	

	pLenOut:POINTER TO UINT;
	pDataOut:POINTER TO BYTE;
END_VAR
VAR
	index: UINT;

	i: INT;
END_VAR

fn_cyber_userdata200 := FALSE;

index := 0;

pDataOut[index] := ANY_TO_BYTE(data0/256/256/256 MOD 256);
index := index + 1;
pDataOut[index] := ANY_TO_BYTE(data0/256/256 MOD 256);
index := index + 1;
pDataOut[index] := ANY_TO_BYTE(data0/256 MOD 256);
index := index + 1;
pDataOut[index] := ANY_TO_BYTE(data0 MOD 256);
index := index + 1;

pDataOut[index] := ANY_TO_BYTE(data1/256/256/256 MOD 256);
index := index + 1;
pDataOut[index] := ANY_TO_BYTE(data1/256/256 MOD 256);
index := index + 1;
pDataOut[index] := ANY_TO_BYTE(data1/256 MOD 256);
index := index + 1;
pDataOut[index] := ANY_TO_BYTE(data1 MOD 256);
index := index + 1;

pDataOut[index] := ANY_TO_BYTE(data2/256/256/256 MOD 256);
index := index + 1;
pDataOut[index] := ANY_TO_BYTE(data2/256/256 MOD 256);
index := index + 1;
pDataOut[index] := ANY_TO_BYTE(data2/256 MOD 256);
index := index + 1;
pDataOut[index] := ANY_TO_BYTE(data2 MOD 256);
index := index + 1;

pDataOut[index] := ANY_TO_BYTE(data3/256/256/256 MOD 256);
index := index + 1;
pDataOut[index] := ANY_TO_BYTE(data3/256/256 MOD 256);
index := index + 1;
pDataOut[index] := ANY_TO_BYTE(data3/256 MOD 256);
index := index + 1;
pDataOut[index] := ANY_TO_BYTE(data3 MOD 256);
index := index + 1;

pDataOut[index] := ANY_TO_BYTE(data4/256/256/256 MOD 256);
index := index + 1;
pDataOut[index] := ANY_TO_BYTE(data4/256/256 MOD 256);
index := index + 1;
pDataOut[index] := ANY_TO_BYTE(data4/256 MOD 256);
index := index + 1;
pDataOut[index] := ANY_TO_BYTE(data4 MOD 256);
index := index + 1;

pDataOut[index] := ANY_TO_BYTE(data5/256/256/256 MOD 256);
index := index + 1;
pDataOut[index] := ANY_TO_BYTE(data5/256/256 MOD 256);
index := index + 1;
pDataOut[index] := ANY_TO_BYTE(data5/256 MOD 256);
index := index + 1;
pDataOut[index] := ANY_TO_BYTE(data5 MOD 256);
index := index + 1;

pDataOut[index] := ANY_TO_BYTE(data6/256/256/256 MOD 256);
index := index + 1;
pDataOut[index] := ANY_TO_BYTE(data6/256/256 MOD 256);
index := index + 1;
pDataOut[index] := ANY_TO_BYTE(data6/256 MOD 256);
index := index + 1;
pDataOut[index] := ANY_TO_BYTE(data6 MOD 256);
index := index + 1;

pDataOut[index] := ANY_TO_BYTE(data7/256/256/256 MOD 256);
index := index + 1;
pDataOut[index] := ANY_TO_BYTE(data7/256/256 MOD 256);
index := index + 1;
pDataOut[index] := ANY_TO_BYTE(data7/256 MOD 256);
index := index + 1;
pDataOut[index] := ANY_TO_BYTE(data7 MOD 256);
index := index + 1;



pLenOut^ := index;

fn_cyber_userdata200 := TRUE;

END_FUNCTION

// MIC7001/Application/GPRS/fb_m26
FUNCTION_BLOCK fb_m26
VAR_INPUT
	enable :BOOL := FALSE;
	ipaddr :STRING(32);
	port :UINT;
END_VAR
VAR_OUTPUT
	xBusy :BOOL := FALSE;
	xError :BOOL := FALSE;
	xDone :BOOL := FALSE;
	handle_m26 :CAA.HANDLE; 
END_VAR
VAR
	udp_init:Udp_Init;
	iStat :UINT := 0;
END_VAR

IF NOT enable THEN
	xBusy := FALSE;
	xError := FALSE;
	handle_m26 := 0;
	RETURN;
END_IF

CASE iStat OF
0:
	udp_init(xExecute := FALSE, ip_addr := ipaddr, port := port);
	udp_init.xExecute := TRUE;
	iStat := 10;
	
10:
	IF udp_init.xDone THEN
		xBusy := TRUE;
		handle_m26 := udp_init.udp_handle;
		iStat := 100;
	ELSIF udp_init.xError THEN
		iStat := 200;
	END_IF	

100:
	xDone:= TRUE;
	
200:
	xError := TRUE;

END_CASE


udp_init(ip_addr := ipaddr, port := port);

END_FUNCTION_BLOCK

// MIC7001/Application/gprs_lib/Udp_Init
FUNCTION_BLOCK Udp_Init
VAR_INPUT
	xExecute:BOOL := FALSE;
	ip_addr:STRING;
	port:UINT;
END_VAR
VAR_OUTPUT
	xDone :BOOL := FALSE;
	xError :BOOL := FALSE;
	xBusy :BOOL := FALSE;
	
	udp_handle :CAA.HANDLE; 
END_VAR
VAR
	udp_config_fb :Udp_Config;
	ComWrite: COM.Write;
	ComRead: COM.Read;	
	com_handle: CAA.HANDLE;
	init_start :DWORD := 0;
	iStat: INT := 0;
END_VAR

init_start := %ID48;
IF (init_start > 0) THEN
	RETURN;
END_IF

IF NOT xExecute THEN
	xDone := FALSE;
	xError := FALSE;
	xBusy := FALSE;
	iStat := 0;
	RETURN;
END_IF

CASE iStat OF
0:
	udp_config_fb(xExecute := FALSE,ip_addr := ip_addr, port := port, com_hand := com_handle); 
	iStat := 10;
	xBusy := TRUE;
10:
	udp_config_fb.xExecute := TRUE;
	IF udp_config_fb.xDone  THEN
		iStat := 100;
		xDone := TRUE;
		xBusy := FALSE;
		udp_handle := com_handle;
		ComWrite(xExecute := FALSE, hCom:= com_handle);
		ComRead(xExecute := FALSE, hCom:= com_handle);		
	ELSIF udp_config_fb.xError THEN
		xError := TRUE;
		iStat := 200;
	END_IF	
100: //succ

200: //error

END_CASE

udp_config_fb(ip_addr := ip_addr, port := port, com_hand := com_handle);

END_FUNCTION_BLOCK

// MIC7001/Application/gprs_lib/Udp_Config
FUNCTION_BLOCK Udp_Config
VAR_INPUT
	xExecute : BOOL := FALSE;
	ip_addr:STRING;
	port:UINT;
END_VAR
VAR_IN_OUT
	com_hand: CAA.HANDLE;
END_VAR
VAR_OUTPUT
	xDone : BOOL := FALSE;
	xError :BOOL := FALSE;
	xBusy : BOOL := FALSE;
END_VAR
VAR
	ton_fb :TON;
	Com1Params: 			ARRAY [1..7] OF COM.PARAMETER;	(* Settings to communicate with 
the COM Port *)
	ComOpen: 				COM.Open;
	ComClose: 				COM.Close;
	ComWrite: 				COM.Write;
	ComRead: 				COM.Read;	
	Rcv_Cnt: 				CAA.SIZE;
	xCom1CloseError: 		BOOL;
	xCom1WriteError: 		BOOL;
	xCom1ReadError: 		BOOL;
	uiComState: INT := 0;
	ComID:USINT:=6;

	position :INT := 0;
	at_cmd :STRING := 'AT$r';
	at_buffer :STRING;
	ate0_cmd :STRING := 'ATE0$r';
	ate0_buffer :STRING;
	cpin_cmd :STRING := 'AT+CPIN?$r';
	cpin_buffer :STRING;
	csq_cmd :STRING := 'AT+CSQ$r';
	csq_buffer :STRING;
	creg_cmd :STRING := 'AT+CREG?$r';
	creg_buffer :STRING;
	cgreg_cmd :STRING := 'AT+CGREG?$r';
	cgreg_buffer :STRING;
	qindi_cmd :STRING := 'AT+QINDI=1$r';
	qindi_buffer :STRING;     
	qimode_cmd :STRING := 'AT+QIMODE=0$r';
	qimode_buffer :STRING;     
	qifgcnt_cmd :STRING := 'AT+QIFGCNT=0$r';
	qifgcnt_buffer :STRING;
	qimux_cmd :STRING := 'AT+QIMUX=0$r';
	qimux_buffer :STRING;
	qicsgp_cmd :STRING := 'AT+QICSGP=1,$"CMNET$"$r';
	qicsgp_buffer :STRING;
	qideact_cmd :STRING := 'AT+QIDEACT$r';
	qideact_buffer :STRING;
	qiregapp_cmd :STRING := 'AT+QIREGAPP$r';
	qiregapp_buffer :STRING;
	qiact_cmd :STRING := 'AT+QIACT$r';
	qiact_buffer :STRING;
	qilocip_cmd :STRING := 'AT+QILOCIP$r';
	qilocip_buffer :STRING;
	qiopen_cmd :STRING := 'AT+QIOPEN=$"UDP$",$"';
	qiopen_buffer :STRING;
	loop_in_count :INT := 0;
	loop_out_count :INT := 0;
	
	reset_gprs_fb :reset_gprs;
END_VAR

IF NOT xExecute THEN
	xDone := FALSE;
	xError := FALSE;
	xBusy := FALSE;
	uiComState := 0;
	RETURN;
END_IF

CASE uiComState OF
	0:
	Com1Params[1].udiParameterId := COM.CAA_Parameter_Constants.udiPort;
	Com1Params[1].udiValue := ComID; 
	Com1Params[2].udiParameterId := COM.CAA_Parameter_Constants.udiBaudrate;
	Com1Params[2].udiValue := 115200;
	Com1Params[3].udiParameterId := COM.CAA_Parameter_Constants.udiParity;
	Com1Params[3].udiValue := INT_TO_UINT(COM.PARITY.NONE);
	Com1Params[4].udiParameterId := COM.CAA_Parameter_Constants.udiStopBits;
	Com1Params[4].udiValue := INT_TO_UINT(COM.STOPBIT.ONESTOPBIT);
	Com1Params[5].udiParameterId := COM.CAA_Parameter_Constants.udiTimeout;
	Com1Params[5].udiValue := 0;
	Com1Params[6].udiParameterId := COM.CAA_Parameter_Constants.udiByteSize;
	Com1Params[6].udiValue := 8;
	Com1Params[7].udiParameterId := COM.CAA_Parameter_Constants.udiBinary;
	Com1Params[7].udiValue := 0;					
	ComOpen(xExecute := TRUE, usiListLength:=UINT_TO_USINT(SIZEOF(Com1Params)/SIZEOF(COM.PARAMETER)),pParameterList:= ADR(Com1Params),hCom=> com_hand);			
	IF ComOpen.xError THEN
		uiComState := 32767;
	ELSIF ComOpen.xDone THEN
		uiComState := 1;
		com_hand := ComOpen.hCom;
		ComWrite(xExecute := FALSE,hCom:= com_hand);	
		ComRead(xExecute := FALSE,hCom:= com_hand);
	END_IF
	
	1:  // write "AT\r"
	ComWrite(xExecute := TRUE,hCom:= com_hand,pBuffer:= ADR(at_cmd),szSize:=len(at_cmd));		
	IF ComWrite.xError THEN
		uiComState := 32767;
	END_IF
	IF ComWrite.xDone THEN
		ComWrite(xExecute := FALSE, hCom:= com_hand);
		uiComState := 2;
	END_IF
	
	2:
	ton_fb(IN := TRUE, PT := TIME#300MS);
	IF (ton_fb.Q) THEN
		ton_fb(IN := FALSE, PT := TIME#300MS);
		uiComState := 3;
	END_IF
	
	3:
	ComRead(xExecute := TRUE,hCom:= com_hand, pBuffer:= ADR(at_buffer), szBuffer:= SIZEOF(at_buffer));			
	IF ComRead.xError THEN
		uiComState := 32767;
	END_IF
	IF ComRead.xDone THEN
		uiComState := 1;
		position := find(at_buffer, 'OK');
		IF position > 0 THEN
			uiComState := 4;
			loop_in_count := 0;
			loop_out_count := 0;
		END_IF
		ComRead(xExecute := FALSE, hCom:= com_hand);
	
		IF loop_out_count > 10 THEN
			uiComState := 32767;
			RETURN;
		END_IF
		
		// 通过gpio复位gprs模块
		loop_in_count := loop_in_count + 1;
		IF loop_in_count > 50 THEN
			loop_in_count := 0;
			loop_out_count := loop_out_count + 1;
			reset_gprs_fb(xExecute := FALSE);
			uiComState := 49;
			RETURN;
		END_IF
	END_IF
		
	4: // write "ATE0\r"
	ComWrite(xExecute := TRUE,hCom:= com_hand,pBuffer:= ADR(ate0_cmd),szSize:=len(ate0_cmd));		
	IF ComWrite.xError THEN
		uiComState := 32767;
	END_IF
	IF ComWrite.xDone THEN
		ComWrite(xExecute := FALSE, hCom:= com_hand);
		uiComState := 5;
	END_IF
	
	5:
	ton_fb(IN := TRUE, PT := TIME#300MS);
	IF (ton_fb.Q) THEN
		ton_fb(IN := FALSE, PT := TIME#300MS);
		uiComState := 6;
	END_IF
	
	6:
	ComRead(xExecute := TRUE,hCom:= com_hand, pBuffer:= ADR(ate0_buffer), szBuffer:= SIZEOF(ate0_buffer));			
	IF ComRead.xError THEN
		uiComState := 32767;
	END_IF
	IF ComRead.xDone THEN
		uiComState := 4;
		ComRead(xExecute := FALSE, hCom:= com_hand);
		position := find(ate0_buffer, 'OK');
		IF position > 0 THEN
			uiComState := 7;
		END_IF
	END_IF
	
	7: // write "AT+CPIN?\r"
	ComWrite(xExecute := TRUE,hCom:= com_hand,pBuffer:= ADR(cpin_cmd),szSize:=len(cpin_cmd));		
	IF ComWrite.xError THEN
		uiComState := 32767;
	END_IF
	IF ComWrite.xDone THEN
		ComWrite(xExecute := FALSE, hCom:= com_hand);
		uiComState := 8;
	END_IF
	
	8:
	ton_fb(IN := TRUE, PT := TIME#300MS);
	IF (ton_fb.Q) THEN
		ton_fb(IN := FALSE, PT := TIME#300MS);
		uiComState := 9;
	END_IF
	
	9:
	ComRead(xExecute := TRUE,hCom:= com_hand, pBuffer:= ADR(cpin_buffer), szBuffer:= SIZEOF(cpin_buffer));			
	IF ComRead.xError THEN
		uiComState := 32767;
	END_IF
	IF ComRead.xDone THEN
		uiComState := 7;
		ComRead(xExecute := FALSE, hCom:= com_hand);
		position := find(cpin_buffer, 'OK');
		IF position > 0 THEN
			uiComState := 10;
		END_IF
	END_IF
	
	10: // write "AT+CSQ\r"
	ComWrite(xExecute := TRUE,hCom:= com_hand,pBuffer:= ADR(csq_cmd),szSize:=len(csq_cmd));		
	IF ComWrite.xError THEN
		uiComState := 32767;
	END_IF
	IF ComWrite.xDone THEN
		ComWrite(xExecute := FALSE, hCom:= com_hand);
		uiComState := 11;
	END_IF
	
	11:
	ton_fb(IN := TRUE, PT := TIME#300MS);
	IF (ton_fb.Q) THEN
		ton_fb(IN := FALSE, PT := TIME#300MS);
		uiComState := 12;
	END_IF
	
	12:
	ComRead(xExecute := TRUE,hCom:= com_hand, pBuffer:= ADR(csq_buffer), szBuffer:= SIZEOF(csq_buffer));			
	IF ComRead.xError THEN
		uiComState := 32767;
	END_IF
	IF ComRead.xDone THEN
		uiComState := 10;
		ComRead(xExecute := FALSE, hCom:= com_hand);
		position := find(csq_buffer, 'OK');
		IF position > 0 THEN
			uiComState := 13;
		END_IF
	END_IF
	
	13: // write "AT+CREG?\r"
	ComWrite(xExecute := TRUE,hCom:= com_hand,pBuffer:= ADR(creg_cmd),szSize:=len(creg_cmd));		
	IF ComWrite.xError THEN
		uiComState := 32767;
	END_IF
	IF ComWrite.xDone THEN
		ComWrite(xExecute := FALSE, hCom:= com_hand);
		uiComState := 14;
	END_IF
	
	14:
	ton_fb(IN := TRUE, PT := TIME#300MS);
	IF (ton_fb.Q) THEN
		ton_fb(IN := FALSE, PT := TIME#300MS);
		uiComState := 15;
	END_IF
	
	15:
	ComRead(xExecute := TRUE,hCom:= com_hand, pBuffer:= ADR(creg_buffer), szBuffer:= SIZEOF(creg_buffer));			
	IF ComRead.xError THEN
		uiComState := 32767;
	END_IF
	IF ComRead.xDone THEN
		uiComState := 13;
		ComRead(xExecute := FALSE, hCom:= com_hand);
		position := find(creg_buffer, 'OK');
		IF position > 0 THEN
			uiComState := 16;
		END_IF
	END_IF
	
	16: // write "AT+CGREG?\r"
	ComWrite(xExecute := TRUE,hCom:= com_hand,pBuffer:= ADR(cgreg_cmd),szSize:=len(cgreg_cmd));		
	IF ComWrite.xError THEN
		uiComState := 32767;
	END_IF
	IF ComWrite.xDone THEN
		ComWrite(xExecute := FALSE, hCom:= com_hand);
		uiComState := 17;
	END_IF
	
	17:
	ton_fb(IN := TRUE, PT := TIME#300MS);
	IF (ton_fb.Q) THEN
		ton_fb(IN := FALSE, PT := TIME#300MS);
		uiComState := 18;
	END_IF
	
	18:
	ComRead(xExecute := TRUE,hCom:= com_hand, pBuffer:= ADR(cgreg_buffer), szBuffer:= SIZEOF(cgreg_buffer));			
	IF ComRead.xError THEN
		uiComState := 32767;
	END_IF
	IF ComRead.xDone THEN
		uiComState := 16;
		ComRead(xExecute := FALSE, hCom:= com_hand);
		position := find(cgreg_buffer, 'OK');
		IF position > 0 THEN
			uiComState := 19;
		END_IF
	END_IF
	
	19: // write "AT+QINDI=1\r"     
	ComWrite(xExecute := TRUE,hCom:= com_hand,pBuffer:= ADR(qindi_cmd),szSize:=len(qindi_cmd));		
	IF ComWrite.xError THEN
		uiComState := 32767;
	END_IF
	IF ComWrite.xDone THEN
		ComWrite(xExecute := FALSE, hCom:= com_hand);
		uiComState := 20;
	END_IF
	
	20:
	ton_fb(IN := TRUE, PT := TIME#300MS);
	IF (ton_fb.Q) THEN
		ton_fb(IN := FALSE, PT := TIME#300MS);
		uiComState := 21;
	END_IF
	
	21:
	ComRead(xExecute := TRUE,hCom:= com_hand, pBuffer:= ADR(qindi_buffer), szBuffer:= SIZEOF(qindi_buffer));			
	IF ComRead.xError THEN
		uiComState := 32767;
	END_IF
	IF ComRead.xDone THEN
		uiComState := 19;
		ComRead(xExecute := FALSE, hCom:= com_hand);
		position := find(qindi_buffer, 'OK');
		IF position > 0 THEN
			uiComState := 22;
			loop_in_count := 0;
			loop_out_count := 0;
		ELSE
			IF loop_out_count > 10 THEN
				uiComState := 32767;
				RETURN;
			END_IF
			
			// 通过gpio复位gprs模块
			loop_in_count := loop_in_count + 1;
			IF loop_in_count > 25 THEN
				loop_in_count := 0;
				loop_out_count := loop_out_count + 1;
				reset_gprs_fb(xExecute := FALSE);
				uiComState := 49;
				RETURN;
			END_IF
		END_IF
	END_IF
	
	22: // write "AT+QIMODE=0\r"     
	ComWrite(xExecute := TRUE,hCom:= com_hand,pBuffer:= ADR(qimode_cmd),szSize:=len(qimode_cmd));		
	IF ComWrite.xError THEN
		uiComState := 32767;
	END_IF
	IF ComWrite.xDone THEN
		ComWrite(xExecute := FALSE, hCom:= com_hand);
		uiComState := 23;
	END_IF
	
	23:
	ton_fb(IN := TRUE, PT := TIME#300MS);
	IF (ton_fb.Q) THEN
		ton_fb(IN := FALSE, PT := TIME#300MS);
		uiComState := 24;
	END_IF
	
	24:
	ComRead(xExecute := TRUE,hCom:= com_hand, pBuffer:= ADR(qimode_buffer), szBuffer:= SIZEOF(qimode_buffer));			
	IF ComRead.xError THEN
		uiComState := 32767;
	END_IF
	IF ComRead.xDone THEN
		uiComState := 22;
		ComRead(xExecute := FALSE, hCom:= com_hand);
		position := find(qimode_buffer, 'OK');
		IF position > 0 THEN
			uiComState := 25;
		ELSE
			IF loop_out_count > 10 THEN
				uiComState := 32767;
				RETURN;
			END_IF
			
			// 通过gpio复位gprs模块
			loop_in_count := loop_in_count + 1;
			IF loop_in_count > 25 THEN
				loop_in_count := 0;
				loop_out_count := loop_out_count + 1;
				reset_gprs_fb(xExecute := FALSE);
				uiComState := 49;
				RETURN;
			END_IF
		END_IF
		//uiComState := 25;
	END_IF
	
	25: // write "AT+QIFGCNT=0\r"     
	ComWrite(xExecute := TRUE,hCom:= com_hand,pBuffer:= ADR(qifgcnt_cmd),szSize:=len(qifgcnt_cmd));		
	IF ComWrite.xError THEN
		uiComState := 32767;
	END_IF
	IF ComWrite.xDone THEN
		ComWrite(xExecute := FALSE, hCom:= com_hand);
		uiComState := 26;
	END_IF
	
	26:
	ton_fb(IN := TRUE, PT := TIME#300MS);
	IF (ton_fb.Q) THEN
		ton_fb(IN := FALSE, PT := TIME#300MS);
		uiComState := 27;
	END_IF
	
	27:
	ComRead(xExecute := TRUE,hCom:= com_hand, pBuffer:= ADR(qifgcnt_buffer), szBuffer:= SIZEOF(qifgcnt_buffer));			
	IF ComRead.xError THEN
		uiComState := 32767;
	END_IF
	IF ComRead.xDone THEN
		uiComState := 25;
		ComRead(xExecute := FALSE, hCom:= com_hand);
		position := find(qifgcnt_buffer, 'OK');
		IF position > 0 THEN
			uiComState := 28;
		END_IF
	END_IF
	
	28: // write "AT+QIMUX=0\r"     
	ComWrite(xExecute := TRUE,hCom:= com_hand,pBuffer:= ADR(qimux_cmd),szSize:=len(qimux_cmd));		
	IF ComWrite.xError THEN
		uiComState := 32767;
	END_IF
	IF ComWrite.xDone THEN
		ComWrite(xExecute := FALSE, hCom:= com_hand);
		uiComState := 29;
	END_IF
	
	29:
	ton_fb(IN := TRUE, PT := TIME#300MS);
	IF (ton_fb.Q) THEN
		ton_fb(IN := FALSE, PT := TIME#300MS);
		uiComState := 30;
	END_IF
	
	30:
	ComRead(xExecute := TRUE,hCom:= com_hand, pBuffer:= ADR(qimux_buffer), szBuffer:= SIZEOF(qimux_buffer));			
	IF ComRead.xError THEN
		uiComState := 32767;
	END_IF
	IF ComRead.xDone THEN
		uiComState := 28;
		ComRead(xExecute := FALSE, hCom:= com_hand);
		position := find(qimux_buffer, 'OK');
		IF position > 0 THEN
			uiComState := 31;
		END_IF
		//uiComState := 31;
	END_IF
	
	31: // write "AT+QICSGP=1,\"CMNET\"\r"     
	ComWrite(xExecute := TRUE,hCom:= com_hand,pBuffer:= ADR(qicsgp_cmd),szSize:=len(qicsgp_cmd));		
	IF ComWrite.xError THEN
		uiComState := 32767;
	END_IF
	IF ComWrite.xDone THEN
		ComWrite(xExecute := FALSE, hCom:= com_hand);
		uiComState := 32;
	END_IF
	
	32:
	ton_fb(IN := TRUE, PT := TIME#300MS);
	IF (ton_fb.Q) THEN
		ton_fb(IN := FALSE, PT := TIME#300MS);
		uiComState := 33;
	END_IF
	
	33:
	ComRead(xExecute := TRUE,hCom:= com_hand, pBuffer:= ADR(qicsgp_buffer), szBuffer:= SIZEOF(qicsgp_buffer));			
	IF ComRead.xError THEN
		uiComState := 32767;
	END_IF
	IF ComRead.xDone THEN
		uiComState := 31;
		ComRead(xExecute := FALSE, hCom:= com_hand);
		position := find(qicsgp_buffer, 'OK');
		IF position > 0 THEN
			uiComState := 34;
		END_IF
	END_IF
	
	34: // write "AT+QIDEACT\r"     
	ComWrite(xExecute := TRUE,hCom:= com_hand,pBuffer:= ADR(qideact_cmd),szSize:=len(qideact_cmd));		
	IF ComWrite.xError THEN
		uiComState := 32767;
	END_IF
	IF ComWrite.xDone THEN
		ComWrite(xExecute := FALSE, hCom:= com_hand);
		uiComState := 35;
	END_IF
	
	35:
	ton_fb(IN := TRUE, PT := TIME#300MS);
	IF (ton_fb.Q) THEN
		ton_fb(IN := FALSE, PT := TIME#300MS);
		uiComState := 36;
	END_IF
	
	36:
	ComRead(xExecute := TRUE,hCom:= com_hand, pBuffer:= ADR(qicsgp_buffer), szBuffer:= SIZEOF(qicsgp_buffer));			
	IF ComRead.xError THEN
		uiComState := 32767;
	END_IF
	IF ComRead.xDone THEN
		uiComState := 34;
		ComRead(xExecute := FALSE, hCom:= com_hand);
		position := find(qicsgp_buffer, 'DEACT OK');
		IF position > 0 THEN
			uiComState := 37;
		END_IF
	END_IF
	
	37: // write "AT+QIREGAPP\r"     
	ComWrite(xExecute := TRUE,hCom:= com_hand,pBuffer:= ADR(qiregapp_cmd),szSize:=len(qiregapp_cmd));		
	IF ComWrite.xError THEN
		uiComState := 32767;
	END_IF
	IF ComWrite.xDone THEN
		ComWrite(xExecute := FALSE, hCom:= com_hand);
		uiComState := 38;
	END_IF
	
	38:
	ton_fb(IN := TRUE, PT := TIME#300MS);
	IF (ton_fb.Q) THEN
		ton_fb(IN := FALSE, PT := TIME#300MS);
		uiComState := 39;
	END_IF
	
	39:
	ComRead(xExecute := TRUE,hCom:= com_hand, pBuffer:= ADR(qiregapp_buffer), szBuffer:= SIZEOF(qiregapp_buffer));			
	IF ComRead.xError THEN
		uiComState := 32767;
	END_IF
	IF ComRead.xDone THEN
		uiComState := 37;
		ComRead(xExecute := FALSE, hCom:= com_hand);
		position := find(qiregapp_buffer, 'OK');
		IF position > 0 THEN
			uiComState := 40;
		END_IF
	END_IF
	
	40: // write "AT+QIACT\r"     
	ComWrite(xExecute := TRUE,hCom:= com_hand,pBuffer:= ADR(qiact_cmd),szSize:=len(qiact_cmd));		
	IF ComWrite.xError THEN
		uiComState := 32767;
	END_IF
	IF ComWrite.xDone THEN
		ComWrite(xExecute := FALSE, hCom:= com_hand);
		uiComState := 41;
	END_IF
	
	41:
	ton_fb(IN := TRUE, PT := TIME#300MS);
	IF (ton_fb.Q) THEN
		ton_fb(IN := FALSE, PT := TIME#300MS);
		uiComState := 42;
	END_IF
	
	42:
	ComRead(xExecute := TRUE,hCom:= com_hand, pBuffer:= ADR(qiact_buffer), szBuffer:= SIZEOF(qiact_buffer));			
	IF ComRead.xError THEN
		uiComState := 32767;
	END_IF
	IF ComRead.xDone THEN
		uiComState := 40;
		ComRead(xExecute := FALSE, hCom:= com_hand);
		position := find(qiact_buffer, 'OK');
		IF position > 0 THEN
			uiComState := 43;
		END_IF
	END_IF
	
	43: // write "AT+QILOCIP\r"     
	ComWrite(xExecute := TRUE,hCom:= com_hand,pBuffer:= ADR(qilocip_cmd),szSize:=len(qilocip_cmd));		
	IF ComWrite.xError THEN
		uiComState := 32767;
	END_IF
	IF ComWrite.xDone THEN
		ComWrite(xExecute := FALSE, hCom:= com_hand);
		uiComState := 44;
	END_IF
	
	44:
	ton_fb(IN := TRUE, PT := TIME#300MS);
	IF (ton_fb.Q) THEN
		ton_fb(IN := FALSE, PT := TIME#300MS);
		uiComState := 45;
	END_IF
	
	45:
	ComRead(xExecute := TRUE,hCom:= com_hand, pBuffer:= ADR(qilocip_buffer), szBuffer:= SIZEOF(qilocip_buffer));			
	IF ComRead.xError THEN
		uiComState := 32767;
	END_IF
	IF ComRead.xDone THEN
		uiComState := 46;
		ComRead(xExecute := FALSE, hCom:= com_hand);
		position := find(qilocip_buffer, 'ERROR');
		IF position > 0 THEN
			uiComState := 43;
		END_IF
	END_IF
	
	46: // write "AT+QIOPEN=\"UDP\",\"47.107.240.29\",123456\r"  
	qiopen_cmd := concat(qiopen_cmd, ip_addr);
	qiopen_cmd := concat(qiopen_cmd, '$",');
	qiopen_cmd := concat(qiopen_cmd, ANY_TO_STRING(port));
	qiopen_cmd := concat(qiopen_cmd, '$r');   
	ComWrite(xExecute := TRUE,hCom:= com_hand,pBuffer:= ADR(qiopen_cmd),szSize:=len(qiopen_cmd));		
	IF ComWrite.xError THEN
		uiComState := 32767;
	END_IF
	IF ComWrite.xDone THEN
		ComWrite(xExecute := FALSE, hCom:= com_hand);
		uiComState := 47;
	END_IF
	
	47:
	ton_fb(IN := TRUE, PT := TIME#300MS);
	IF (ton_fb.Q) THEN
		ton_fb(IN := FALSE, PT := TIME#300MS);
		uiComState := 48;
	END_IF
	
	48:
	ComRead(xExecute := TRUE,hCom:= com_hand, pBuffer:= ADR(qiopen_buffer), szBuffer:= SIZEOF(qiopen_buffer));			
	IF ComRead.xError THEN
		uiComState := 32767;
	END_IF
	IF ComRead.xDone THEN
		uiComState := 46;
		ComRead(xExecute := FALSE, hCom:= com_hand);
		position := find(qiopen_buffer, 'CONNECT OK');
		IF position > 0 THEN
			uiComState := 255;
		ELSE
			position := find(qiopen_buffer, 'ALREAY CONNECT');
			IF position > 0 THEN
				uiComState := 255;
			END_IF
		END_IF
	END_IF
	
	49:
	reset_gprs_fb.xExecute := TRUE;
	IF reset_gprs_fb.xDone THEN
		uiComState := 1;
	END_IF
	
	255:
		xDone := TRUE;
		
	32767:	
		xError := TRUE;
END_CASE

reset_gprs_fb();

END_FUNCTION_BLOCK

// MIC7001/Application/gprs_lib/reset_gprs
FUNCTION_BLOCK reset_gprs
VAR_INPUT
	xExecute:BOOL := FALSE;
END_VAR
VAR_OUTPUT
	xDone : BOOL := FALSE;
	xError :BOOL := FALSE;
	xBusy :BOOL := FALSE;
END_VAR
VAR
	iState :INT := 0;
	ton_fb :TON; 
END_VAR

IF NOT xExecute THEN
	iState := 0;
	xDone := FALSE;
	xBusy := FALSE;
	xError := FALSE;
	RETURN;
END_IF

CASE iState OF
0:
	xBusy := TRUE;
	set_gpio_value(129, 1);
	iState := 10;
	
10:
	ton_fb(IN := TRUE, PT := TIME#2000MS);
	IF (ton_fb.Q) THEN
		ton_fb(IN := FALSE, PT := TIME#2000MS);
		iState := 20;
	END_IF
	
20:
	set_gpio_value(129, 0);
	iState := 30;
	
30:
	ton_fb(IN := TRUE, PT := TIME#5000MS);
	IF (ton_fb.Q) THEN
		ton_fb(IN := FALSE, PT := TIME#5000MS);
		iState := 40;
	END_IF
	
40:
	iState := 255;	
	
255:
	xDone := TRUE;
	xBusy := FALSE;
32767:
	xError := TRUE;
END_CASE

END_FUNCTION_BLOCK

// MIC7001/Application/gprs_lib/Udp_Write
FUNCTION_BLOCK Udp_Write
VAR_INPUT
	xExecute :BOOL := FALSE;
	com :CAA.HANDLE;
	buffer: CAA.PVOID;
	size :CAA.SIZE;
END_VAR
VAR_OUTPUT
	xDone :BOOL := FALSE;
	xBusy :BOOL := FALSE;
	xError :BOOL := FALSE;
	atcState :INT;
END_VAR
VAR
	ComWrite: COM.Write;
	ComRead: COM.Read;	
	qisend_buffer :STRING := 'AT+QISEND='; 
	ton_fb :TON;  
	ack_buffer1 :STRING;
	ack_buffer2 :STRING;
	position :INT := -1;
	end_flag :ARRAY[0..1] OF BYTE;
	actionState :INT := 0;
	loop_count1 :INT := 0;
	loop_count2 :INT := 0;
	read_data_buffer: ARRAY[0..1499] OF BYTE;
END_VAR

IF NOT xExecute OR com = 0 THEN
	xDone := FALSE;
	xError := FALSE;
	xBusy := FALSE;
	actionState := 0;
	qisend_buffer := 'AT+QISEND='; 
	ComWrite(xExecute := FALSE);
	ComRead(xExecute := FALSE);
	RETURN;
END_IF

CASE actionState OF
0:
	ComRead(xExecute := TRUE,hCom:= com, pBuffer:= ADR(read_data_buffer), szBuffer:= SIZEOF(read_data_buffer));			
	IF ComRead.xError THEN
		ComRead(xExecute := FALSE);		
		actionState := 32767;
	END_IF
	IF ComRead.xDone THEN
		ComRead(xExecute := FALSE);			
		actionState := 1;
	END_IF

1:
	qisend_buffer := concat(qisend_buffer, ANY_TO_STRING(size));
	qisend_buffer := concat(qisend_buffer, '$r'); 
	actionState := 5;
	
5:
	ComWrite(xExecute := TRUE, hCom:= com, pBuffer:= ADR(qisend_buffer), szSize:= len(qisend_buffer));
	IF ComWrite.xError THEN
		actionState := 32767;
	END_IF
	IF ComWrite.xDone THEN
		actionState := 10;
		ComWrite(xExecute := FALSE, hCom:= com);	
	END_IF
	
10:
	ton_fb(IN := TRUE, PT := TIME#200MS);
	IF (ton_fb.Q) THEN
		ton_fb(IN := FALSE, PT := TIME#200MS);
		actionState := 20;
		ComRead(xExecute := FALSE);		
	END_IF
	
20:
	ComRead(xExecute := TRUE,hCom:= com, pBuffer:= ADR(ack_buffer1), szBuffer:= SIZEOF(ack_buffer1));			
	IF ComRead.xError THEN
		atcState := 32767;
	END_IF
	IF ComRead.xDone THEN
		
		position := find(ack_buffer1, '>');
		IF position > 0 THEN
			actionState := 30;
		ELSE
			actionState := 10;
		END_IF
		ComRead(xExecute := FALSE, hCom:= com);
		
		loop_count1 := loop_count1 + 1;
		IF loop_count1 > 50 THEN
			loop_count1 := 0;
			actionState := 32767;
		END_IF
	END_IF
	
30:
	ComWrite(xExecute := TRUE, hCom:= com, pBuffer:= buffer, szSize:= size);
	IF ComWrite.xError THEN
		actionState := 32767;
	END_IF
	IF ComWrite.xDone THEN
		actionState := 40;
		ComWrite(xExecute := FALSE, hCom:= com);	
	END_IF
	
40:
	end_flag[0] := 16#1A;
	ComWrite(xExecute := TRUE, hCom:= com, pBuffer:= ADR(end_flag), szSize:= 1);
	IF ComWrite.xError THEN
		actionState := 32767;
	END_IF
	IF ComWrite.xDone THEN
		actionState := 50;
		ComWrite(xExecute := FALSE, hCom:= com);	
	END_IF
	
50:
	ton_fb(IN := TRUE, PT := TIME#300MS);
	IF (ton_fb.Q) THEN
		ton_fb(IN := FALSE, PT := TIME#300MS);
		actionState := 60;
	END_IF
	
60:
	ComRead(xExecute := TRUE,hCom:= com, pBuffer:= ADR(ack_buffer2), szBuffer:= SIZEOF(ack_buffer2));			
	IF ComRead.xError THEN
		atcState := 32767;
	END_IF
	IF ComRead.xDone THEN
		position := find(ack_buffer2, 'SEND OK');
		IF position > 0 THEN
			actionState := 255;
		ELSE
			actionState := 50;
		END_IF
		ComRead(xExecute := FALSE, hCom:= com);
		loop_count2 := loop_count2 + 1;
		IF loop_count2 > 50 THEN
			loop_count2 := 0;
			actionState := 32767;
		END_IF
	END_IF
	
255:
	xDone := TRUE;
	xError := FALSE;
	xBusy := FALSE;
	actionState := 250;

	loop_count1 := 0;
	loop_count2 := 0; 
	ack_buffer1 := '';
	ack_buffer2 := '';
	qisend_buffer := 'AT+QISEND=';	
	
250:

32767:
	xDone := FALSE;
	xError := TRUE;
	xBusy := FALSE;
	actionState := 32700;

	loop_count1 := 0;
	loop_count2 := 0; 
	ack_buffer1 := '';
	ack_buffer2 := '';
	qisend_buffer := 'AT+QISEND=';	
	
32700:

END_CASE

END_FUNCTION_BLOCK

// MIC7001/Application/gprs_lib/UDP_Read
FUNCTION_BLOCK UDP_Read
VAR_INPUT
	xExecute:BOOL := FALSE;
	com :CAA.HANDLE;
	buffer: CAA.PVOID;
	rsize : CAA.SIZE;
END_VAR
VAR_OUTPUT
	xDone :BOOL := FALSE;
	xBusy :BOOL := FALSE;
	xError :BOOL := FALSE;
	size :CAA.SIZE;
	
END_VAR
VAR
	ton_fb :TON;  
	ComWrite: COM.Write;
	ComRead: COM.Read;	
	ack_buffer :STRING[1499];
	//ack_buffer :ARRAY[0..1499] OF BYTE;
	position :INT := -1;
	qird :STRING := 'AT+QIRD=0,1,0,1500$R';

	read_data_buffer: ARRAY[0..1499] OF BYTE;
	read_tmp_buffer: ARRAY[0..1499] OF BYTE;
	i :INT;
	read_num :INT;
	comma1 :INT;
	comma2 :INT;
	new_line :INT;
	data_len :INT := 0;
	//uchar *pos, *comma1, *comma2, *new_line;
	
	loop_count :INT := 0;
	loop_exit :INT := 0;
	
	del_atcState :INT;
	iStat :UINT := 0;
END_VAR

IF com = 0 OR NOT xExecute THEN
	xDone := FALSE;
	xError := FALSE;
	xBusy := FALSE;
	iStat := 0;
	position := -1;
	size := 0;
	ComRead(xExecute := FALSE);
	RETURN;
END_IF

CASE iStat OF
	0:
	ComRead(xExecute := TRUE,hCom:= com, pBuffer:= ADR(ack_buffer), szBuffer:= SIZEOF(ack_buffer));			
	IF ComRead.xError THEN
		ComRead(xExecute := FALSE, hCom:= com);
		iStat := 32767;
	END_IF
	
	IF ComRead.xDone THEN
		position := find(ack_buffer, '+QIRDI: 0,1,0');
		IF position > 0 THEN
			iStat := 2;
		ELSE
			iStat := 1;
		END_IF
		ComRead(xExecute := FALSE, hCom:= com);
		loop_count := loop_count + 1;
		IF loop_count > 20 THEN
			iStat := 2;
			loop_count := 0;
		END_IF
	END_IF
	
	1:
	ton_fb(IN := TRUE, PT := TIME#300MS);
	IF (ton_fb.Q) THEN
		ton_fb(IN := FALSE, PT := TIME#300MS);
		iStat := 0;
	END_IF
	
	2:
	ComWrite(xExecute := TRUE, hCom:= com, pBuffer:= ADR(qird), szSize:= len(qird));
	IF ComWrite.xError THEN
		iStat := 32767;
	END_IF
	
	IF ComWrite.xDone THEN
		iStat := 3;
		ComWrite(xExecute := FALSE, hCom:= com);	
	END_IF
	
	3:
	ton_fb(IN := TRUE, PT := TIME#300MS);
	IF (ton_fb.Q) THEN
		ton_fb(IN := FALSE, PT := TIME#300MS);
		iStat := 4;
	END_IF
	
	4:
	ComRead(xExecute := TRUE,hCom:= com, pBuffer:= ADR(read_data_buffer), szBuffer:= rsize);			
	IF ComRead.xError THEN
		iStat := 32767;
	END_IF
	IF ComRead.xDone THEN
		iStat := 5;
		read_num :=  ANY_TO_INT(ComRead.szSize);
		ComRead(xExecute := FALSE, hCom:= com);		
	END_IF
	
	5: //查找第一个逗号，第二次读取的时候，会返回OK，表示已经读完
	IF read_num = 6 THEN
		iStat := 0;
		loop_exit := loop_exit + 1;
		IF loop_exit > 1 THEN
			loop_exit := 0;
			iStat := 32767;
		END_IF
		RETURN;
	END_IF
	FOR i := 0 TO read_num - 1 BY 1 DO
		iStat := 32767;
		IF read_data_buffer[i] = 16#2C THEN
			comma1 := i;
			iStat := 6;
			RETURN;
		END_IF
	END_FOR;
	
	6: //查找第二个逗号
	FOR i := comma1 + 1 TO read_num - 1 BY 1 DO
		iStat := 32767;
		IF read_data_buffer[i] = 16#2C THEN
			comma2 := i;
			iStat := 7;
			RETURN;
		END_IF
	END_FOR;
	
	7: //查找回车换行
	FOR i := comma2 + 1 TO read_num - 1 BY 1 DO
		iStat := 32767;
		IF read_data_buffer[i] = 16#0D  AND read_data_buffer[i + 1] = 16#0A THEN
			new_line := i;
			iStat := 8;
			RETURN;
		END_IF
	END_FOR;
	
	8: // 获取数据长度
	FOR i := comma2 + 1 TO new_line - 1 BY 1 DO
		data_len := data_len *10 + read_data_buffer[i] - 16#30;
	END_FOR;

	iStat := 255;
	IF data_len > 0 THEN
		size := data_len;
		SysMemCpy(pDest:=buffer,pSrc:=ADR(read_data_buffer) + new_line + 2, udiCount:=data_len);
		
		data_len := 0;
		ack_buffer := '';
		loop_count := 0;
		read_num := 0;
		FOR i := 0 TO 1499 BY 1 DO
			read_data_buffer[i] := 0;
		END_FOR
	END_IF
	
	255:
		ComRead(xExecute := FALSE);
		xDone := TRUE;
		xBusy := FALSE;
		xError := FALSE;
		iStat := 256;
		
		data_len := 0;
		ack_buffer := '';
		loop_count := 0;
		read_num := 0;
		FOR i := 0 TO 1499 BY 1 DO
			read_data_buffer[i] := 0;
		END_FOR		
	256:
	
	32767:
		ComRead(xExecute := FALSE);
		xError := TRUE;
		xDone := FALSE;
		xBusy := FALSE;
		iStat := 32700;
		
		data_len := 0;
		ack_buffer := '';
		loop_count := 0;
		read_num := 0;
		FOR i := 0 TO 1499 BY 1 DO
			read_data_buffer[i] := 0;
		END_FOR		
	32700:
	
END_CASE

END_FUNCTION_BLOCK

// MIC7001/Application/GPRS/File_Read
FUNCTION_BLOCK File_Read
VAR_INPUT
	file_name :STRING;
END_VAR
VAR_OUTPUT
	sReadLine		: STRING;
	isRead          :BOOL := FALSE;	
END_VAR
VAR
	hfile			: CAA.HANDLE;
	FileOpen 		: File.Open;
	FileClose		: File.Close;
	FileRead		: File.Read;
	
	iState			: UINT := 0;	
	xError			: BOOL := FALSE;
END_VAR

 CASE iState OF
	0: // Open the file again, with read access.
	   isRead := false;
	   FileOpen(xExecute:= TRUE, sFileName:= file_name, xExclusive:= FALSE, eFileMode:= File.MODE.MREAD);
	   IF FileOpen.xDone = TRUE THEN
		   hfile := FileOpen.hFile;
		   FileOpen(xExecute:= FALSE);
		   iState := 1;
		   sReadLine := '';
	   ELSIF FileOpen.xError = TRUE THEN
		   iState:= 32767;
		   FileOpen(xExecute:= FALSE);
	   END_IF

	1: // Read the string from the file.
	   FileRead(xExecute:= TRUE, hFile:= hfile, pBuffer:= ADR(sReadLine), szBuffer:= SIZEOF(sReadLine));
	   IF FileRead.xDone = TRUE THEN
		   iState := 2;		   
		   sReadLine := MID(sReadLine, ANY_TO_INT(FileRead.szSize), 1);
		   FileRead(xExecute:= FALSE);
	   ELSIF FileRead.xError = TRUE THEN
		   iState:= 32767;
		   FileRead(xExecute:= FALSE);
	   END_IF 
	   
	 2: // Close that file.
	   FileClose(xExecute:= TRUE, hFile:= hfile);
	   IF FileClose.xDone = TRUE THEN
		   iState := 3;
		   FileClose(xExecute:= FALSE);
	   ELSIF FileClose.xError = TRUE THEN
		   iState:= 32767;
		   FileClose(xExecute:= FALSE);
	   END_IF
	   
	3: 	  
		isRead := TRUE;
		iState := 0;
		
	32767: 		
	
END_CASE

END_FUNCTION_BLOCK

// MIC7001/Application/gprs_lib/Com_Read
FUNCTION_BLOCK Com_Read
VAR_INPUT
	xExecute:BOOL := FALSE;
	com :CAA.HANDLE;
	wbuffer: CAA.PVOID;
	wsize :CAA.SIZE;	
	rbuffer: CAA.PVOID;
	rsize : CAA.SIZE;
END_VAR
VAR_OUTPUT
	xDone:BOOL := FALSE;
	xBusy:BOOL := FALSE;
	xError:BOOL := FALSE;
	size :CAA.SIZE;
END_VAR
VAR
	iState :INT;
	ton_fb :TON;  
	ComWrite: COM.Write;
	ComRead: COM.Read;	
	actionState :INT;
END_VAR

IF NOT xExecute THEN
	iState := 0;
	xDone := FALSE;
	xBusy := FALSE;
	xError := FALSE;
	size := 0;
	RETURN;
END_IF

CASE iState OF
0:
	size := 0;
	ComWrite(xExecute := TRUE, hCom:= com, pBuffer:= wbuffer, szSize:= wsize);
	IF ComWrite.xError THEN
		iState := 32767;
	END_IF
	IF ComWrite.xDone THEN
		iState := 10;
		ComWrite(xExecute := FALSE, hCom:= com);	
	END_IF
	xBusy := TRUE;
	
10:
	ton_fb(IN := TRUE, PT := TIME#300MS);
	IF (ton_fb.Q) THEN
		ton_fb(IN := FALSE, PT := TIME#300MS);
		iState := 20;
	END_IF
	
20:
	ComRead(xExecute := TRUE,hCom:= com, pBuffer:= rbuffer, szBuffer:= rsize);			
	IF ComRead.xError THEN
		iState := 32767;
	END_IF
	IF ComRead.xDone THEN
		iState := 255;
		size := ComRead.szSize;
		ComRead(xExecute := FALSE, hCom:= com);		
	END_IF
	
255:
	xDone := TRUE;
	xBusy := FALSE;
	
32767:
	xError := TRUE;
	
END_CASE

END_FUNCTION_BLOCK

// MIC7001/Application/GPRS/fb_get_iccid
FUNCTION_BLOCK fb_get_iccid
VAR_INPUT
	xExecute:BOOL := FALSE;
	m26_handle:CAA.HANDLE; 
END_VAR

VAR_OUTPUT
	iccid:STRING(32);
	xDone:BOOL := FALSE;
	xBusy :BOOL := FALSE;
	xError:BOOL := FALSE;
END_VAR

VAR
	iStat:UINT := 0;
	udp_handle :CAA.HANDLE; 
	accid_cmd :STRING := 'AT+ICCID$r';
	iccid_read_buffer :STRING(255);
	com_read :Com_Read;
	udp_init_fb: INT;
	size:CAA.SIZE;
	position :INT := -1;
	ICCID_HEAD:STRING := '+ICCID: ';
	timer01:ton;
END_VAR


IF NOT xExecute OR m26_handle = 0 THEN
	xDone := FALSE;
	xBusy := FALSE;
	xError := FALSE;
	iccid := '';
	iStat := 0;
	RETURN;
END_IF 		

IF iccid <> '' THEN  //已经读到了，不需再读
	xDone := TRUE;
	xBusy := FALSE;
	xError := FALSE;
	RETURN; 
END_IF

CASE iStat OF
0:
	com_read(xExecute := FALSE);
	iStat := 10;
	timer01(in := FALSE);
	com_read.xExecute := TRUE;
10:
	IF com_read.xDone THEN
		IF com_read.size > 0 THEN
			position := find(iccid_read_buffer, ICCID_HEAD);
			IF position > 0 THEN
				iccid := mid(iccid_read_buffer, 20, position + len(ICCID_HEAD));
				xDone := TRUE;
				iStat := 100;
			END_IF
		END_IF
	ELSIF com_read.xError THEN
		xDone := FALSE;
		iStat := 200;
	END_IF	
	timer01(in := NOT timer01.Q, pt := T#2S);
	IF timer01.Q THEN
		iStat := 0;
	END_IF
100:

200:

END_CASE

com_read(com:= m26_handle, wbuffer:= ADR(accid_cmd), wsize := len(accid_cmd), rbuffer := ADR(iccid_read_buffer), rsize := SIZEOF(iccid_read_buffer));

END_FUNCTION_BLOCK

// MIC7001/Application/GPRS/fb_get_lac
FUNCTION_BLOCK fb_get_lac
VAR_INPUT
	xExecute:BOOL := FALSE;
	m26_handle:CAA.HANDLE; 
END_VAR
VAR_OUTPUT
	lac:STRING(4) := '0000';
	ci :STRING(4) := '0000';
	xDone:BOOL := FALSE;
	xError:BOOL := FALSE;
END_VAR
VAR
	iStat:UINT := 0;
	udp_handle :CAA.HANDLE; 
	lac_set_cmd :STRING := 'AT+CREG=2$r';
	lac_get_cmd :STRING := 'AT+CREG?$r';
	lac_close_cmd :STRING := 'AT+CREG=0$r';
	lac_read_buffer :STRING(255);
	com_read :Com_Read;
	udp_init_fb: INT;
	size:CAA.SIZE;
	position :INT := -1;
	LACID_HEAD:STRING := '+CREG:';
	lac_str:STRING(8);
	ci_str:STRING(8);
	cntr: INT;
END_VAR


IF m26_handle = 0 THEN
	RETURN;
END_IF

IF NOT xExecute THEN
	xDone := FALSE;
	xError := FALSE;
	lac := '0000';
	ci := '0000';
	iStat := 0;
	
	RETURN;
END_IF 		

CASE iStat OF
0:
	com_read(xExecute := FALSE);
	com_read.wbuffer:= ADR(lac_set_cmd);
 	com_read.wsize := len(lac_set_cmd);
	com_read.xExecute := TRUE;	
	iStat := 5;
5:  //set m26 for lac and ci with command:  AT+CREG=2
	IF com_read.xDone THEN
		size := com_read.size;
		IF size > 0 THEN
			position := find(lac_read_buffer, 'OK');
			IF position > 0 THEN
				com_read(xExecute := FALSE);
				com_read.wbuffer:= ADR(lac_get_cmd);
				com_read.wsize := len(lac_get_cmd);
				com_read.xExecute := TRUE;				
				iStat := 10;
				cntr := 0;
			END_IF
		ELSE
			iStat := 0;
		END_IF
	ELSIF com_read.xError THEN
		xDone := FALSE;
	END_IF	

10:  //read lac and ci with command: AT+CREG?
	IF com_read.xDone THEN
		IF com_read.size > 0 THEN
			position := find(lac_read_buffer, LACID_HEAD);
			IF position > 0 THEN
				position := find(lac_read_buffer, '$"');
				IF position > 0 THEN
					lac := mid(lac_read_buffer, 4, position + 1);
					ci := mid(lac_read_buffer, 4, position + 8);
					iStat := 20;
					size := 0;
					com_read(xExecute := FALSE);
					com_read.wbuffer:= ADR(lac_close_cmd);
 					com_read.wsize := len(lac_close_cmd);
					com_read.xExecute := TRUE;
				END_IF
			ELSE
				iStat := 0;
			END_IF
		END_IF
		cntr := cntr + 1;
		IF cntr > 50 THEN
			iStat := 0;
		END_IF
	ELSIF com_read.xError THEN
		xDone := FALSE;
	END_IF	
	
20:  //close
	IF com_read.xDone THEN
		size := com_read.size;
		IF size > 0 THEN
			position := find(lac_read_buffer, 'OK');
			IF position > 0 THEN
				iStat := 100;
				xDone := TRUE;
			END_IF
		ELSE
			xDone := FALSE;
		END_IF
	ELSIF com_read.xError THEN
		xDone := FALSE;
	END_IF	
100: //ok

END_CASE

com_read(com:= m26_handle, rbuffer := ADR(lac_read_buffer), rsize := SIZEOF(lac_read_buffer));

END_FUNCTION_BLOCK
